LIN {X 0,Y 418.639,Z 217.334,A -85,B 0,C 180,E1 -10080,E2 -10080} C_VEL
LIN {X 0,Y 418.468,Z 217.355,A -85,B 0,C 180,E1 -10082.888,E2 -10082.888} C_VEL
LIN {X 0,Y 418.469,Z 217.355,A -85,B 0,C 180,E1 -10085.783,E2 -10085.783} C_VEL
LIN {X 0,Y 418.35,Z 217.368,A -85,B 0,C 180,E1 -10088.696,E2 -10088.696} C_VEL
LIN {X 0,Y 418.299,Z 217.373,A -85,B 0,C 180,E1 -10091.631,E2 -10091.631} C_VEL
LIN {X 0,Y 418.273,Z 217.382,A -85,B 0,C 180,E1 -10094.598,E2 -10094.598} C_VEL
LIN {X 0,Y 418.252,Z 217.38,A -85,B 0,C 180,E1 -10097.605,E2 -10097.605} C_VEL
LIN {X 0,Y 418.223,Z 217.388,A -85,B 0,C 180,E1 -10100.664,E2 -10100.664} C_VEL
LIN {X 0,Y 418.248,Z 217.383,A -85,B 0,C 180,E1 -10103.784,E2 -10103.784} C_VEL
LIN {X 0,Y 418.203,Z 217.392,A -85,B 0,C 180,E1 -10107.049,E2 -10107.049} C_VEL
LIN {X 0,Y 418.219,Z 217.385,A -85,B 0,C 180,E1 -10110.274,E2 -10110.274} C_VEL
LIN {X 0,Y 418.213,Z 217.383,A -85,B 0,C 180,E1 -10113.68,E2 -10113.68} C_VEL
LIN {X 0,Y 418.221,Z 217.379,A -85,B 0,C 180,E1 -10117.226,E2 -10117.226} C_VEL
LIN {X 0,Y 418.219,Z 217.379,A -85,B 0,C 180,E1 -10119.686,E2 -10119.686} C_VEL
LIN {X 0,Y 418.214,Z 217.391,A -85,B 0,C 180,E1 -10122.322,E2 -10122.322} C_VEL
LIN {X 0,Y 418.223,Z 217.385,A -85,B 0,C 180,E1 -10125.11,E2 -10125.11} C_VEL
LIN {X 0,Y 418.221,Z 217.386,A -85,B 0,C 180,E1 -10127.767,E2 -10127.767} C_VEL
LIN {X 0,Y 418.23,Z 217.385,A -85,B 0,C 180,E1 -10131.558,E2 -10131.558} C_VEL
LIN {X 0,Y 418.254,Z 217.383,A -85,B 0,C 180,E1 -10135.16,E2 -10135.16} C_VEL
LIN {X 0,Y 418.241,Z 217.384,A -85,B 0,C 180,E1 -10137.473,E2 -10137.473} C_VEL
LIN {X 0,Y 418.292,Z 217.381,A -85,B 0,C 180,E1 -10141.146,E2 -10141.146} C_VEL
LIN {X 0,Y 418.302,Z 217.657,A -85,B 0,C 180,E1 -10141.33,E2 -10141.33} C_VEL
LIN {X 0,Y 421.008,Z 229.949,A -85,B 0,C 180,E1 -10144.012,E2 -10144.012} C_VEL
LIN {X 0,Y 421.849,Z 235.282,A -85,B 0,C 180,E1 -10145.124,E2 -10145.124} C_VEL
LIN {X 0,Y 420.782,Z 249.932,A -85,B 0,C 180,E1 -10147.927,E2 -10147.927} C_VEL
LIN {X 0,Y 419.911,Z 263.738,A -85,B 0,C 180,E1 -10150.533,E2 -10150.533} C_VEL
LIN {X 0,Y 423.774,Z 286.188,A -85,B 0,C 180,E1 -10151.146,E2 -10151.146} C_VEL
LIN {X 0,Y 424.458,Z 292.992,A -85,B 0,C 180,E1 -10151.303,E2 -10151.303} C_VEL
LIN {X 0,Y 423.498,Z 373.222,A -85,B 0,C 180,E1 -10152.713,E2 -10152.713} C_VEL
LIN {X 0,Y 422.871,Z 386.948,A -85,B 0,C 180,E1 -10153.153,E2 -10153.153} C_VEL
LIN {X 0,Y 422.143,Z 399.294,A -85,B 0,C 180,E1 -10153.745,E2 -10153.745} C_VEL
LIN {X 0,Y 421.315,Z 411.136,A -85,B 0,C 180,E1 -10154.52,E2 -10154.52} C_VEL
LIN {X 0,Y 420.483,Z 422.531,A -85,B 0,C 180,E1 -10155.48,E2 -10155.48} C_VEL
LIN {X 0,Y 419.616,Z 432.832,A -85,B 0,C 180,E1 -10156.562,E2 -10156.562} C_VEL
LIN {X 0,Y 419.038,Z 441.272,A -85,B 0,C 180,E1 -10157.652,E2 -10157.652} C_VEL
LIN {X 0,Y 418.232,Z 450.447,A -85,B 0,C 180,E1 -10159.102,E2 -10159.102} C_VEL
LIN {X 0,Y 417.726,Z 457.856,A -85,B 0,C 180,E1 -10160.558,E2 -10160.558} C_VEL
LIN {X 0,Y 417.325,Z 464.7,A -85,B 0,C 180,E1 -10162.256,E2 -10162.256} C_VEL
LIN {X 0,Y 417.123,Z 469.362,A -85,B 0,C 180,E1 -10163.762,E2 -10163.762} C_VEL
LIN {X 0,Y 417.104,Z 472.691,A -85,B 0,C 180,E1 -10165.166,E2 -10165.166} C_VEL
LIN {X 0,Y 417.069,Z 475.74,A -85,B 0,C 180,E1 -10167.101,E2 -10167.101} C_VEL
LIN {X 0,Y 417.091,Z 476.67,A -85,B 0,C 180,E1 -10168.067,E2 -10168.067} C_VEL
LIN {X 0,Y 417.058,Z 477.19,A -85,B 0,C 180,E1 -10169.033,E2 -10169.033} C_VEL
LIN {X 0,Y 417.056,Z 477.282,A -85,B 0,C 180,E1 -10169.998,E2 -10169.998} C_VEL
LIN {X 0,Y 417.092,Z 476.305,A -85,B 0,C 180,E1 -10171.929,E2 -10171.929} C_VEL
LIN {X 0,Y 417.102,Z 475.215,A -85,B 0,C 180,E1 -10172.895,E2 -10172.895} C_VEL
LIN {X 0,Y 417.023,Z 473.664,A -85,B 0,C 180,E1 -10173.863,E2 -10173.863} C_VEL
LIN {X 0,Y 417.13,Z 470.551,A -85,B 0,C 180,E1 -10175.315,E2 -10175.315} C_VEL
LIN {X 0,Y 417.229,Z 466.36,A -85,B 0,C 180,E1 -10176.769,E2 -10176.769} C_VEL
LIN {X 0,Y 417.45,Z 459.955,A -85,B 0,C 180,E1 -10178.468,E2 -10178.468} C_VEL
LIN {X 0,Y 417.798,Z 452.974,A -85,B 0,C 180,E1 -10179.926,E2 -10179.926} C_VEL
LIN {X 0,Y 418.226,Z 445.837,A -85,B 0,C 180,E1 -10181.14,E2 -10181.14} C_VEL
LIN {X 0,Y 418.747,Z 437.203,A -85,B 0,C 180,E1 -10182.353,E2 -10182.353} C_VEL
LIN {X 0,Y 419.452,Z 426.544,A -85,B 0,C 180,E1 -10183.563,E2 -10183.563} C_VEL
LIN {X 0,Y 420.103,Z 415.971,A -85,B 0,C 180,E1 -10184.53,E2 -10184.53} C_VEL
LIN {X 0,Y 420.782,Z 404.288,A -85,B 0,C 180,E1 -10185.372,E2 -10185.372} C_VEL
LIN {X 0,Y 421.426,Z 392.137,A -85,B 0,C 180,E1 -10186.031,E2 -10186.031} C_VEL
LIN {X 0,Y 421.967,Z 379.849,A -85,B 0,C 180,E1 -10186.506,E2 -10186.506} C_VEL
LIN {X 0,Y 422.292,Z 366.152,A -85,B 0,C 180,E1 -10186.835,E2 -10186.835} C_VEL
LIN {X 0,Y 422.863,Z 289.846,A -85,B 0,C 180,E1 -10188.135,E2 -10188.135} C_VEL
LIN {X 0,Y 419.286,Z 264.116,A -85,B 0,C 180,E1 -10188.725,E2 -10188.725} C_VEL
LIN {X 0,Y 420.277,Z 245.887,A -85,B 0,C 180,E1 -10192.097,E2 -10192.097} C_VEL
LIN {X 0,Y 421.029,Z 232.178,A -85,B 0,C 180,E1 -10194.66,E2 -10194.66} C_VEL
LIN {X 0,Y 419.604,Z 223.737,A -85,B 0,C 180,E1 -10196.345,E2 -10196.345} C_VEL
LIN {X 0,Y 418.339,Z 217.378,A -85,B 0,C 180,E1 -10197.69,E2 -10197.69} C_VEL
LIN {X 0,Y 418.195,Z 217.393,A -85,B 0,C 180,E1 -10201.392,E2 -10201.392} C_VEL
LIN {X 0,Y 418.246,Z 217.384,A -85,B 0,C 180,E1 -10204.576,E2 -10204.576} C_VEL
LIN {X 0,Y 418.205,Z 217.393,A -85,B 0,C 180,E1 -10207.829,E2 -10207.829} C_VEL
LIN {X 0,Y 418.196,Z 217.389,A -85,B 0,C 180,E1 -10210.944,E2 -10210.944} C_VEL
LIN {X 0,Y 418.182,Z 217.396,A -85,B 0,C 180,E1 -10213.725,E2 -10213.725} C_VEL
LIN {X 0,Y 418.231,Z 217.385,A -85,B 0,C 180,E1 -10216.451,E2 -10216.451} C_VEL
LIN {X 0,Y 418.234,Z 217.385,A -85,B 0,C 180,E1 -10219.119,E2 -10219.119} C_VEL
LIN {X 0,Y 418.202,Z 217.39,A -85,B 0,C 180,E1 -10222.161,E2 -10222.161} C_VEL
LIN {X 0,Y 418.226,Z 217.389,A -85,B 0,C 180,E1 -10225.416,E2 -10225.416} C_VEL
LIN {X 0,Y 418.173,Z 217.391,A -85,B 0,C 180,E1 -10228.601,E2 -10228.601} C_VEL
LIN {X 0,Y 418.251,Z 217.385,A -85,B 0,C 180,E1 -10231.934,E2 -10231.934} C_VEL
LIN {X 0,Y 418.245,Z 217.386,A -85,B 0,C 180,E1 -10235.16,E2 -10235.16} C_VEL
LIN {X 0,Y 418.225,Z 217.385,A -85,B 0,C 180,E1 -10238.303,E2 -10238.303} C_VEL
LIN {X 0,Y 418.239,Z 217.391,A -85,B 0,C 180,E1 -10241.381,E2 -10241.381} C_VEL
LIN {X 0,Y 418.259,Z 217.381,A -85,B 0,C 180,E1 -10244.404,E2 -10244.404} C_VEL
LIN {X 0,Y 418.319,Z 217.379,A -85,B 0,C 180,E1 -10247.385,E2 -10247.385} C_VEL
LIN {X 0,Y 418.364,Z 217.374,A -85,B 0,C 180,E1 -10251.304,E2 -10251.304} C_VEL
LIN {X 0,Y 418.486,Z 217.352,A -85,B 0,C 180,E1 -10254.217,E2 -10254.217} C_VEL
LIN {X 0,Y 418.489,Z 217.352,A -85,B 0,C 180,E1 -10258.075,E2 -10258.075} C_VEL
LIN {X 0,Y 418.616,Z 217.336,A -85,B 0,C 180,E1 -10260,E2 -10260} C_VEL
LIN {X 0,Y 418.446,Z 217.364,A -85,B 0,C 180,E1 -10262.888,E2 -10262.888} C_VEL
LIN {X 0,Y 418.435,Z 217.364,A -85,B 0,C 180,E1 -10266.752,E2 -10266.752} C_VEL
LIN {X 0,Y 418.292,Z 217.377,A -85,B 0,C 180,E1 -10269.673,E2 -10269.673} C_VEL
LIN {X 0,Y 418.304,Z 217.38,A -85,B 0,C 180,E1 -10273.007,E2 -10273.007} C_VEL
LIN {X 0,Y 418.269,Z 217.387,A -85,B 0,C 180,E1 -10276.74,E2 -10276.74} C_VEL
LIN {X 0,Y 418.221,Z 217.386,A -85,B 0,C 180,E1 -10279.792,E2 -10279.792} C_VEL
LIN {X 0,Y 418.185,Z 217.396,A -85,B 0,C 180,E1 -10282.739,E2 -10282.739} C_VEL
LIN {X 0,Y 418.225,Z 217.386,A -85,B 0,C 180,E1 -10285.907,E2 -10285.907} C_VEL
LIN {X 0,Y 418.231,Z 217.385,A -85,B 0,C 180,E1 -10289.165,E2 -10289.165} C_VEL
LIN {X 0,Y 418.217,Z 217.389,A -85,B 0,C 180,E1 -10292.847,E2 -10292.847} C_VEL
LIN {X 0,Y 418.208,Z 217.392,A -85,B 0,C 180,E1 -10296.242,E2 -10296.242} C_VEL
LIN {X 0,Y 418.228,Z 217.385,A -85,B 0,C 180,E1 -10299.685,E2 -10299.685} C_VEL
LIN {X 0,Y 418.252,Z 217.389,A -85,B 0,C 180,E1 -10302.333,E2 -10302.333} C_VEL
LIN {X 0,Y 418.217,Z 217.386,A -85,B 0,C 180,E1 -10305.114,E2 -10305.114} C_VEL
LIN {X 0,Y 418.214,Z 217.389,A -85,B 0,C 180,E1 -10307.771,E2 -10307.771} C_VEL
LIN {X 0,Y 418.234,Z 217.386,A -85,B 0,C 180,E1 -10310.623,E2 -10310.623} C_VEL
LIN {X 0,Y 418.223,Z 217.391,A -85,B 0,C 180,E1 -10313.98,E2 -10313.98} C_VEL
LIN {X 0,Y 418.24,Z 217.383,A -85,B 0,C 180,E1 -10317.16,E2 -10317.16} C_VEL
LIN {X 0,Y 418.255,Z 217.381,A -85,B 0,C 180,E1 -10320.9,E2 -10320.9} C_VEL
LIN {X 0,Y 418.257,Z 217.386,A -85,B 0,C 180,E1 -10324.1,E2 -10324.1} C_VEL
LIN {X 0,Y 418.223,Z 217.386,A -85,B 0,C 180,E1 -10327.267,E2 -10327.267} C_VEL
LIN {X 0,Y 418.277,Z 217.38,A -85,B 0,C 180,E1 -10330.368,E2 -10330.368} C_VEL
LIN {X 0,Y 418.312,Z 217.377,A -85,B 0,C 180,E1 -10333.408,E2 -10333.408} C_VEL
LIN {X 0,Y 418.345,Z 217.371,A -85,B 0,C 180,E1 -10337.002,E2 -10337.002} C_VEL
LIN {X 0,Y 418.362,Z 217.476,A -85,B 0,C 180,E1 -10339.996,E2 -10339.996} C_VEL
LIN {X 0,Y 419.753,Z 225.468,A -85,B 0,C 180,E1 -10341.821,E2 -10341.821} C_VEL
LIN {X 0,Y 419.713,Z 228.011,A -85,B 0,C 180,E1 -10342.371,E2 -10342.371} C_VEL
LIN {X 0,Y 423.404,Z 248.524,A -85,B 0,C 180,E1 -10342.881,E2 -10342.881} C_VEL
LIN {X 0,Y 422.273,Z 335.092,A -85,B 0,C 180,E1 -10344.361,E2 -10344.361} C_VEL
LIN {X 0,Y 421.932,Z 348.28,A -85,B 0,C 180,E1 -10344.776,E2 -10344.776} C_VEL
LIN {X 0,Y 421.84,Z 354.693,A -85,B 0,C 180,E1 -10345.056,E2 -10345.056} C_VEL
LIN {X 0,Y 420.996,Z 360.232,A -85,B 0,C 180,E1 -10345.312,E2 -10345.312} C_VEL
LIN {X 0,Y 417.843,Z 369.054,A -85,B 0,C 180,E1 -10345.756,E2 -10345.756} C_VEL
LIN {X 0,Y 414.563,Z 377.579,A -85,B 0,C 180,E1 -10346.292,E2 -10346.292} C_VEL
LIN {X 0,Y 413.511,Z 382.59,A -85,B 0,C 180,E1 -10346.701,E2 -10346.701} C_VEL
LIN {X 0,Y 412.792,Z 393.404,A -85,B 0,C 180,E1 -10347.807,E2 -10347.807} C_VEL
LIN {X 0,Y 412.144,Z 403.005,A -85,B 0,C 180,E1 -10349.025,E2 -10349.025} C_VEL
LIN {X 0,Y 411.629,Z 410.879,A -85,B 0,C 180,E1 -10350.246,E2 -10350.246} C_VEL
LIN {X 0,Y 411.019,Z 418.618,A -85,B 0,C 180,E1 -10351.716,E2 -10351.716} C_VEL
LIN {X 0,Y 410.69,Z 425.692,A -85,B 0,C 180,E1 -10353.435,E2 -10353.435} C_VEL
LIN {X 0,Y 410.351,Z 430.439,A -85,B 0,C 180,E1 -10354.914,E2 -10354.914} C_VEL
LIN {X 0,Y 410.226,Z 434.196,A -85,B 0,C 180,E1 -10356.453,E2 -10356.453} C_VEL
LIN {X 0,Y 410.057,Z 436.704,A -85,B 0,C 180,E1 -10357.882,E2 -10357.882} C_VEL
LIN {X 0,Y 409.974,Z 437.947,A -85,B 0,C 180,E1 -10358.876,E2 -10358.876} C_VEL
LIN {X 0,Y 409.907,Z 438.765,A -85,B 0,C 180,E1 -10359.873,E2 -10359.873} C_VEL
LIN {X 0,Y 409.966,Z 439.155,A -85,B 0,C 180,E1 -10360.87,E2 -10360.87} C_VEL
LIN {X 0,Y 410,Z 439.052,A -85,B 0,C 180,E1 -10362.294,E2 -10362.294} C_VEL
LIN {X 0,Y 410.021,Z 437.952,A -85,B 0,C 180,E1 -10363.885,E2 -10363.885} C_VEL
LIN {X 0,Y 410.108,Z 436.698,A -85,B 0,C 180,E1 -10364.896,E2 -10364.896} C_VEL
LIN {X 0,Y 410.413,Z 433.881,A -85,B 0,C 180,E1 -10366.471,E2 -10366.471} C_VEL
LIN {X 0,Y 410.681,Z 430.238,A -85,B 0,C 180,E1 -10367.941,E2 -10367.941} C_VEL
LIN {X 0,Y 411.096,Z 425.31,A -85,B 0,C 180,E1 -10369.464,E2 -10369.464} C_VEL
LIN {X 0,Y 411.684,Z 418.963,A -85,B 0,C 180,E1 -10371.008,E2 -10371.008} C_VEL
LIN {X 0,Y 412.304,Z 412.445,A -85,B 0,C 180,E1 -10372.288,E2 -10372.288} C_VEL
LIN {X 0,Y 413.037,Z 404.552,A -85,B 0,C 180,E1 -10373.569,E2 -10373.569} C_VEL
LIN {X 0,Y 413.863,Z 394.792,A -85,B 0,C 180,E1 -10374.852,E2 -10374.852} C_VEL
LIN {X 0,Y 414.764,Z 384.155,A -85,B 0,C 180,E1 -10375.974,E2 -10375.974} C_VEL
LIN {X 0,Y 415.548,Z 373.203,A -85,B 0,C 180,E1 -10376.898,E2 -10376.898} C_VEL
LIN {X 0,Y 416.144,Z 361.394,A -85,B 0,C 180,E1 -10377.672,E2 -10377.672} C_VEL
LIN {X 0,Y 416.778,Z 348.137,A -85,B 0,C 180,E1 -10378.301,E2 -10378.301} C_VEL
LIN {X 0,Y 417.168,Z 334.958,A -85,B 0,C 180,E1 -10378.713,E2 -10378.713} C_VEL
LIN {X 0,Y 418.332,Z 247.723,A -85,B 0,C 180,E1 -10380.255,E2 -10380.255} C_VEL
LIN {X 0,Y 414.124,Z 230.945,A -85,B 0,C 180,E1 -10380.806,E2 -10380.806} C_VEL
LIN {X 0,Y 413.352,Z 228.534,A -85,B 0,C 180,E1 -10380.923,E2 -10380.923} C_VEL
LIN {X 0,Y 411.227,Z 218.261,A -85,B 0,C 180,E1 -10383.445,E2 -10383.445} C_VEL
LIN {X 0,Y 411.188,Z 218.268,A -85,B 0,C 180,E1 -10386.74,E2 -10386.74} C_VEL
LIN {X 0,Y 411.219,Z 218.263,A -85,B 0,C 180,E1 -10389.728,E2 -10389.728} C_VEL
LIN {X 0,Y 411.168,Z 218.268,A -85,B 0,C 180,E1 -10393.131,E2 -10393.131} C_VEL
LIN {X 0,Y 411.21,Z 218.265,A -85,B 0,C 180,E1 -10395.872,E2 -10395.872} C_VEL
LIN {X 0,Y 411.197,Z 218.264,A -85,B 0,C 180,E1 -10398.763,E2 -10398.763} C_VEL
LIN {X 0,Y 411.188,Z 218.265,A -85,B 0,C 180,E1 -10402.025,E2 -10402.025} C_VEL
LIN {X 0,Y 411.189,Z 218.264,A -85,B 0,C 180,E1 -10405.665,E2 -10405.665} C_VEL
LIN {X 0,Y 411.178,Z 218.261,A -85,B 0,C 180,E1 -10409.151,E2 -10409.151} C_VEL
LIN {X 0,Y 411.24,Z 218.252,A -85,B 0,C 180,E1 -10412.521,E2 -10412.521} C_VEL
LIN {X 0,Y 411.199,Z 218.261,A -85,B 0,C 180,E1 -10415.783,E2 -10415.783} C_VEL
LIN {X 0,Y 411.172,Z 218.265,A -85,B 0,C 180,E1 -10418.964,E2 -10418.964} C_VEL
LIN {X 0,Y 411.228,Z 218.259,A -85,B 0,C 180,E1 -10422.084,E2 -10422.084} C_VEL
LIN {X 0,Y 411.236,Z 218.253,A -85,B 0,C 180,E1 -10425.146,E2 -10425.146} C_VEL
LIN {X 0,Y 411.256,Z 218.252,A -85,B 0,C 180,E1 -10428.166,E2 -10428.166} C_VEL
LIN {X 0,Y 411.418,Z 218.233,A -85,B 0,C 180,E1 -10432.185,E2 -10432.185} C_VEL
LIN {X 0,Y 411.451,Z 218.227,A -85,B 0,C 180,E1 -10434.118,E2 -10434.118} C_VEL
LIN {X 0,Y 411.48,Z 218.22,A -85,B 0,C 180,E1 -10438.042,E2 -10438.042} C_VEL
LIN {X 0,Y 411.61,Z 218.21,A -85,B 0,C 180,E1 -10440,E2 -10440} C_VEL
LIN {X 0,Y 411.425,Z 218.232,A -85,B 0,C 180,E1 -10442.937,E2 -10442.937} C_VEL
LIN {X 0,Y 411.402,Z 218.237,A -85,B 0,C 180,E1 -10446.868,E2 -10446.868} C_VEL
LIN {X 0,Y 411.267,Z 218.252,A -85,B 0,C 180,E1 -10449.839,E2 -10449.839} C_VEL
LIN {X 0,Y 411.283,Z 218.251,A -85,B 0,C 180,E1 -10453.106,E2 -10453.106} C_VEL
LIN {X 0,Y 411.243,Z 218.254,A -85,B 0,C 180,E1 -10456.889,E2 -10456.889} C_VEL
LIN {X 0,Y 411.186,Z 218.263,A -85,B 0,C 180,E1 -10459.989,E2 -10459.989} C_VEL
LIN {X 0,Y 411.171,Z 218.267,A -85,B 0,C 180,E1 -10463.149,E2 -10463.149} C_VEL
LIN {X 0,Y 411.165,Z 218.263,A -85,B 0,C 180,E1 -10466.386,E2 -10466.386} C_VEL
LIN {X 0,Y 411.176,Z 218.26,A -85,B 0,C 180,E1 -10469.715,E2 -10469.715} C_VEL
LIN {X 0,Y 411.186,Z 218.259,A -85,B 0,C 180,E1 -10473.158,E2 -10473.158} C_VEL
LIN {X 0,Y 411.175,Z 218.262,A -85,B 0,C 180,E1 -10476.554,E2 -10476.554} C_VEL
LIN {X 0,Y 411.185,Z 218.255,A -85,B 0,C 180,E1 -10479.727,E2 -10479.727} C_VEL
LIN {X 0,Y 411.159,Z 218.266,A -85,B 0,C 180,E1 -10483.136,E2 -10483.136} C_VEL
LIN {X 0,Y 411.156,Z 218.268,A -85,B 0,C 180,E1 -10485.883,E2 -10485.883} C_VEL
LIN {X 0,Y 411.143,Z 218.267,A -85,B 0,C 180,E1 -10488.775,E2 -10488.775} C_VEL
LIN {X 0,Y 411.179,Z 218.263,A -85,B 0,C 180,E1 -10492.027,E2 -10492.027} C_VEL
LIN {X 0,Y 411.201,Z 218.265,A -85,B 0,C 180,E1 -10495.668,E2 -10495.668} C_VEL
LIN {X 0,Y 411.186,Z 218.267,A -85,B 0,C 180,E1 -10499.153,E2 -10499.153} C_VEL
LIN {X 0,Y 411.247,Z 218.297,A -85,B 0,C 180,E1 -10500.932,E2 -10500.932} C_VEL
LIN {X 0,Y 414.089,Z 231.233,A -85,B 0,C 180,E1 -10503.815,E2 -10503.815} C_VEL
LIN {X 0,Y 414.974,Z 236.561,A -85,B 0,C 180,E1 -10504.951,E2 -10504.951} C_VEL
LIN {X 0,Y 413.866,Z 251.201,A -85,B 0,C 180,E1 -10507.801,E2 -10507.801} C_VEL
LIN {X 0,Y 413.06,Z 263.345,A -85,B 0,C 180,E1 -10510.138,E2 -10510.138} C_VEL
LIN {X 0,Y 417.187,Z 287.154,A -85,B 0,C 180,E1 -10510.811,E2 -10510.811} C_VEL
LIN {X 0,Y 417.832,Z 294.371,A -85,B 0,C 180,E1 -10510.977,E2 -10510.977} C_VEL
LIN {X 0,Y 416.85,Z 372.337,A -85,B 0,C 180,E1 -10512.365,E2 -10512.365} C_VEL
LIN {X 0,Y 416.249,Z 385.481,A -85,B 0,C 180,E1 -10512.782,E2 -10512.782} C_VEL
LIN {X 0,Y 415.49,Z 397.575,A -85,B 0,C 180,E1 -10513.351,E2 -10513.351} C_VEL
LIN {X 0,Y 414.587,Z 409.813,A -85,B 0,C 180,E1 -10514.136,E2 -10514.136} C_VEL
LIN {X 0,Y 413.709,Z 421.384,A -85,B 0,C 180,E1 -10515.111,E2 -10515.111} C_VEL
LIN {X 0,Y 412.805,Z 431.82,A -85,B 0,C 180,E1 -10516.21,E2 -10516.21} C_VEL
LIN {X 0,Y 412.085,Z 441.247,A -85,B 0,C 180,E1 -10517.44,E2 -10517.44} C_VEL
LIN {X 0,Y 411.249,Z 450.358,A -85,B 0,C 180,E1 -10518.915,E2 -10518.915} C_VEL
LIN {X 0,Y 410.701,Z 457.722,A -85,B 0,C 180,E1 -10520.395,E2 -10520.395} C_VEL
LIN {X 0,Y 410.267,Z 464.51,A -85,B 0,C 180,E1 -10522.122,E2 -10522.122} C_VEL
LIN {X 0,Y 410.043,Z 469.447,A -85,B 0,C 180,E1 -10523.775,E2 -10523.775} C_VEL
LIN {X 0,Y 410.012,Z 472.437,A -85,B 0,C 180,E1 -10525.082,E2 -10525.082} C_VEL
LIN {X 0,Y 409.966,Z 475.458,A -85,B 0,C 180,E1 -10527.05,E2 -10527.05} C_VEL
LIN {X 0,Y 410.018,Z 476.376,A -85,B 0,C 180,E1 -10528.034,E2 -10528.034} C_VEL
LIN {X 0,Y 409.98,Z 476.869,A -85,B 0,C 180,E1 -10529.016,E2 -10529.016} C_VEL
LIN {X 0,Y 409.976,Z 476.948,A -85,B 0,C 180,E1 -10529.998,E2 -10529.998} C_VEL
LIN {X 0,Y 410.02,Z 475.945,A -85,B 0,C 180,E1 -10531.963,E2 -10531.963} C_VEL
LIN {X 0,Y 410,Z 474.828,A -85,B 0,C 180,E1 -10532.946,E2 -10532.946} C_VEL
LIN {X 0,Y 409.942,Z 473.261,A -85,B 0,C 180,E1 -10533.93,E2 -10533.93} C_VEL
LIN {X 0,Y 410.025,Z 470.116,A -85,B 0,C 180,E1 -10535.407,E2 -10535.407} C_VEL
LIN {X 0,Y 410.16,Z 465.895,A -85,B 0,C 180,E1 -10536.886,E2 -10536.886} C_VEL
LIN {X 0,Y 410.377,Z 459.453,A -85,B 0,C 180,E1 -10538.616,E2 -10538.616} C_VEL
LIN {X 0,Y 410.736,Z 452.422,A -85,B 0,C 180,E1 -10540.098,E2 -10540.098} C_VEL
LIN {X 0,Y 411.326,Z 443.601,A -85,B 0,C 180,E1 -10541.579,E2 -10541.579} C_VEL
LIN {X 0,Y 411.917,Z 434.557,A -85,B 0,C 180,E1 -10542.812,E2 -10542.812} C_VEL
LIN {X 0,Y 412.601,Z 424.611,A -85,B 0,C 180,E1 -10543.918,E2 -10543.918} C_VEL
LIN {X 0,Y 413.285,Z 413.595,A -85,B 0,C 180,E1 -10544.901,E2 -10544.901} C_VEL
LIN {X 0,Y 414.057,Z 401.237,A -85,B 0,C 180,E1 -10545.755,E2 -10545.755} C_VEL
LIN {X 0,Y 414.688,Z 388.182,A -85,B 0,C 180,E1 -10546.425,E2 -10546.425} C_VEL
LIN {X 0,Y 415.212,Z 374.897,A -85,B 0,C 180,E1 -10546.878,E2 -10546.878} C_VEL
LIN {X 0,Y 415.54,Z 354.224,A -85,B 0,C 180,E1 -10547.276,E2 -10547.276} C_VEL
LIN {X 0,Y 416.04,Z 290.792,A -85,B 0,C 180,E1 -10548.374,E2 -10548.374} C_VEL
LIN {X 0,Y 412.325,Z 263.698,A -85,B 0,C 180,E1 -10549.021,E2 -10549.021} C_VEL
LIN {X 0,Y 413.471,Z 243.924,A -85,B 0,C 180,E1 -10552.745,E2 -10552.745} C_VEL
LIN {X 0,Y 414.039,Z 232.94,A -85,B 0,C 180,E1 -10554.837,E2 -10554.837} C_VEL
LIN {X 0,Y 411.874,Z 221.104,A -85,B 0,C 180,E1 -10557.261,E2 -10557.261} C_VEL
LIN {X 0,Y 411.296,Z 218.255,A -85,B 0,C 180,E1 -10557.884,E2 -10557.884} C_VEL
LIN {X 0,Y 411.165,Z 218.268,A -85,B 0,C 180,E1 -10561.279,E2 -10561.279} C_VEL
LIN {X 0,Y 411.187,Z 218.265,A -85,B 0,C 180,E1 -10564.329,E2 -10564.329} C_VEL
LIN {X 0,Y 411.171,Z 218.271,A -85,B 0,C 180,E1 -10567.97,E2 -10567.97} C_VEL
LIN {X 0,Y 411.137,Z 218.269,A -85,B 0,C 180,E1 -10571.224,E2 -10571.224} C_VEL
LIN {X 0,Y 411.152,Z 218.267,A -85,B 0,C 180,E1 -10574.486,E2 -10574.486} C_VEL
LIN {X 0,Y 411.196,Z 218.262,A -85,B 0,C 180,E1 -10577.293,E2 -10577.293} C_VEL
LIN {X 0,Y 411.197,Z 218.26,A -85,B 0,C 180,E1 -10580.773,E2 -10580.773} C_VEL
LIN {X 0,Y 411.161,Z 218.265,A -85,B 0,C 180,E1 -10584.467,E2 -10584.467} C_VEL
LIN {X 0,Y 411.168,Z 218.264,A -85,B 0,C 180,E1 -10586.87,E2 -10586.87} C_VEL
LIN {X 0,Y 411.198,Z 218.26,A -85,B 0,C 180,E1 -10590.639,E2 -10590.639} C_VEL
LIN {X 0,Y 411.195,Z 218.267,A -85,B 0,C 180,E1 -10593.616,E2 -10593.616} C_VEL
LIN {X 0,Y 411.225,Z 218.263,A -85,B 0,C 180,E1 -10597.333,E2 -10597.333} C_VEL
LIN {X 0,Y 411.219,Z 218.259,A -85,B 0,C 180,E1 -10600.028,E2 -10600.028} C_VEL
LIN {X 0,Y 411.215,Z 218.263,A -85,B 0,C 180,E1 -10603.129,E2 -10603.129} C_VEL
LIN {X 0,Y 411.262,Z 218.255,A -85,B 0,C 180,E1 -10606.89,E2 -10606.89} C_VEL
LIN {X 0,Y 411.261,Z 218.253,A -85,B 0,C 180,E1 -10610.161,E2 -10610.161} C_VEL
LIN {X 0,Y 411.425,Z 218.239,A -85,B 0,C 180,E1 -10613.133,E2 -10613.133} C_VEL
LIN {X 0,Y 411.264,Z 218.259,A -85,B 0,C 180,E1 -10615.099,E2 -10615.099} C_VEL
LIN {X 0,Y 411.459,Z 218.228,A -85,B 0,C 180,E1 -10618.042,E2 -10618.042} C_VEL
LIN {X 0,Y 411.586,Z 218.212,A -85,B 0,C 180,E1 -10620,E2 -10620} C_VEL
LIN {X 0,Y 411.403,Z 218.241,A -85,B 0,C 180,E1 -10622.938,E2 -10622.938} C_VEL
LIN {X 0,Y 411.403,Z 218.242,A -85,B 0,C 180,E1 -10626.868,E2 -10626.868} C_VEL
LIN {X 0,Y 411.245,Z 218.255,A -85,B 0,C 180,E1 -10629.84,E2 -10629.84} C_VEL
LIN {X 0,Y 411.263,Z 218.256,A -85,B 0,C 180,E1 -10633.11,E2 -10633.11} C_VEL
LIN {X 0,Y 411.212,Z 218.264,A -85,B 0,C 180,E1 -10636.891,E2 -10636.891} C_VEL
LIN {X 0,Y 411.162,Z 218.265,A -85,B 0,C 180,E1 -10639.99,E2 -10639.99} C_VEL
LIN {X 0,Y 411.15,Z 218.268,A -85,B 0,C 180,E1 -10643.151,E2 -10643.151} C_VEL
LIN {X 0,Y 411.194,Z 218.266,A -85,B 0,C 180,E1 -10646.384,E2 -10646.384} C_VEL
LIN {X 0,Y 411.168,Z 218.264,A -85,B 0,C 180,E1 -10649.716,E2 -10649.716} C_VEL
LIN {X 0,Y 411.168,Z 218.265,A -85,B 0,C 180,E1 -10653.16,E2 -10653.16} C_VEL
LIN {X 0,Y 411.156,Z 218.271,A -85,B 0,C 180,E1 -10656.556,E2 -10656.556} C_VEL
LIN {X 0,Y 411.191,Z 218.262,A -85,B 0,C 180,E1 -10659.734,E2 -10659.734} C_VEL
LIN {X 0,Y 411.187,Z 218.262,A -85,B 0,C 180,E1 -10663.132,E2 -10663.132} C_VEL
LIN {X 0,Y 411.143,Z 218.27,A -85,B 0,C 180,E1 -10665.885,E2 -10665.885} C_VEL
LIN {X 0,Y 411.139,Z 218.269,A -85,B 0,C 180,E1 -10668.776,E2 -10668.776} C_VEL
LIN {X 0,Y 411.184,Z 218.266,A -85,B 0,C 180,E1 -10671.836,E2 -10671.836} C_VEL
LIN {X 0,Y 411.192,Z 218.261,A -85,B 0,C 180,E1 -10675.126,E2 -10675.126} C_VEL
LIN {X 0,Y 411.149,Z 218.274,A -85,B 0,C 180,E1 -10678.007,E2 -10678.007} C_VEL
LIN {X 0,Y 411.204,Z 218.261,A -85,B 0,C 180,E1 -10681.414,E2 -10681.414} C_VEL
LIN {X 0,Y 411.225,Z 218.261,A -85,B 0,C 180,E1 -10683.623,E2 -10683.623} C_VEL
LIN {X 0,Y 411.187,Z 218.262,A -85,B 0,C 180,E1 -10686.856,E2 -10686.856} C_VEL
LIN {X 0,Y 411.208,Z 218.263,A -85,B 0,C 180,E1 -10690.054,E2 -10690.054} C_VEL
LIN {X 0,Y 411.259,Z 218.254,A -85,B 0,C 180,E1 -10693.135,E2 -10693.135} C_VEL
LIN {X 0,Y 411.304,Z 218.247,A -85,B 0,C 180,E1 -10696.899,E2 -10696.899} C_VEL
LIN {X 0,Y 411.289,Z 218.281,A -85,B 0,C 180,E1 -10699.791,E2 -10699.791} C_VEL
LIN {X 0,Y 412.79,Z 227.061,A -85,B 0,C 180,E1 -10701.822,E2 -10701.822} C_VEL
LIN {X 0,Y 412.784,Z 228.347,A -85,B 0,C 180,E1 -10702.103,E2 -10702.103} C_VEL
LIN {X 0,Y 416.563,Z 248.374,A -85,B 0,C 180,E1 -10702.611,E2 -10702.611} C_VEL
LIN {X 0,Y 415.433,Z 336.2,A -85,B 0,C 180,E1 -10704.146,E2 -10704.146} C_VEL
LIN {X 0,Y 415.025,Z 349.897,A -85,B 0,C 180,E1 -10704.597,E2 -10704.597} C_VEL
LIN {X 0,Y 414.582,Z 362.183,A -85,B 0,C 180,E1 -10705.201,E2 -10705.201} C_VEL
LIN {X 0,Y 414.109,Z 373.942,A -85,B 0,C 180,E1 -10705.988,E2 -10705.988} C_VEL
LIN {X 0,Y 413.511,Z 382.59,A -85,B 0,C 180,E1 -10706.701,E2 -10706.701} C_VEL
LIN {X 0,Y 412.449,Z 387.494,A -85,B 0,C 180,E1 -10707.139,E2 -10707.139} C_VEL
LIN {X 0,Y 409.071,Z 395.155,A -85,B 0,C 180,E1 -10707.887,E2 -10707.887} C_VEL
LIN {X 0,Y 405.808,Z 402.316,A -85,B 0,C 180,E1 -10708.735,E2 -10708.735} C_VEL
LIN {X 0,Y 404.931,Z 406.409,A -85,B 0,C 180,E1 -10709.322,E2 -10709.322} C_VEL
LIN {X 0,Y 404.355,Z 414.744,A -85,B 0,C 180,E1 -10710.749,E2 -10710.749} C_VEL
LIN {X 0,Y 403.843,Z 421.787,A -85,B 0,C 180,E1 -10712.246,E2 -10712.246} C_VEL
LIN {X 0,Y 403.506,Z 428.202,A -85,B 0,C 180,E1 -10713.996,E2 -10713.996} C_VEL
LIN {X 0,Y 403.26,Z 432.454,A -85,B 0,C 180,E1 -10715.502,E2 -10715.502} C_VEL
LIN {X 0,Y 403.056,Z 435.653,A -85,B 0,C 180,E1 -10717.012,E2 -10717.012} C_VEL
LIN {X 0,Y 402.96,Z 437.247,A -85,B 0,C 180,E1 -10718.022,E2 -10718.022} C_VEL
LIN {X 0,Y 402.867,Z 438.429,A -85,B 0,C 180,E1 -10719.034,E2 -10719.034} C_VEL
LIN {X 0,Y 402.883,Z 439.509,A -85,B 0,C 180,E1 -10721.064,E2 -10721.064} C_VEL
LIN {X 0,Y 402.932,Z 439.373,A -85,B 0,C 180,E1 -10722.375,E2 -10722.375} C_VEL
LIN {X 0,Y 402.947,Z 438.114,A -85,B 0,C 180,E1 -10724.134,E2 -10724.134} C_VEL
LIN {X 0,Y 403.076,Z 436.81,A -85,B 0,C 180,E1 -10725.162,E2 -10725.162} C_VEL
LIN {X 0,Y 403.378,Z 434.213,A -85,B 0,C 180,E1 -10726.612,E2 -10726.612} C_VEL
LIN {X 0,Y 403.696,Z 430.14,A -85,B 0,C 180,E1 -10728.262,E2 -10728.262} C_VEL
LIN {X 0,Y 404.145,Z 425.384,A -85,B 0,C 180,E1 -10729.73,E2 -10729.73} C_VEL
LIN {X 0,Y 404.795,Z 418.602,A -85,B 0,C 180,E1 -10731.383,E2 -10731.383} C_VEL
LIN {X 0,Y 405.633,Z 410.532,A -85,B 0,C 180,E1 -10732.924,E2 -10732.924} C_VEL
LIN {X 0,Y 406.421,Z 401.988,A -85,B 0,C 180,E1 -10734.248,E2 -10734.248} C_VEL
LIN {X 0,Y 407.341,Z 391.575,A -85,B 0,C 180,E1 -10735.552,E2 -10735.552} C_VEL
LIN {X 0,Y 408.278,Z 381.135,A -85,B 0,C 180,E1 -10736.586,E2 -10736.586} C_VEL
LIN {X 0,Y 409.074,Z 369.623,A -85,B 0,C 180,E1 -10737.497,E2 -10737.497} C_VEL
LIN {X 0,Y 409.697,Z 357.839,A -85,B 0,C 180,E1 -10738.216,E2 -10738.216} C_VEL
LIN {X 0,Y 410.242,Z 345.167,A -85,B 0,C 180,E1 -10738.765,E2 -10738.765} C_VEL
LIN {X 0,Y 410.609,Z 332.42,A -85,B 0,C 180,E1 -10739.118,E2 -10739.118} C_VEL
LIN {X 0,Y 411.785,Z 249.064,A -85,B 0,C 180,E1 -10740.606,E2 -10740.606} C_VEL
LIN {X 0,Y 407.9,Z 233.47,A -85,B 0,C 180,E1 -10741.13,E2 -10741.13} C_VEL
LIN {X 0,Y 406.258,Z 228.88,A -85,B 0,C 180,E1 -10741.343,E2 -10741.343} C_VEL
LIN {X 0,Y 404.197,Z 219.136,A -85,B 0,C 180,E1 -10743.806,E2 -10743.806} C_VEL
LIN {X 0,Y 404.143,Z 219.146,A -85,B 0,C 180,E1 -10747.49,E2 -10747.49} C_VEL
LIN {X 0,Y 404.158,Z 219.14,A -85,B 0,C 180,E1 -10750.081,E2 -10750.081} C_VEL
LIN {X 0,Y 404.149,Z 219.142,A -85,B 0,C 180,E1 -10753.083,E2 -10753.083} C_VEL
LIN {X 0,Y 404.185,Z 219.141,A -85,B 0,C 180,E1 -10755.931,E2 -10755.931} C_VEL
LIN {X 0,Y 404.151,Z 219.142,A -85,B 0,C 180,E1 -10758.639,E2 -10758.639} C_VEL
LIN {X 0,Y 404.147,Z 219.143,A -85,B 0,C 180,E1 -10761.489,E2 -10761.489} C_VEL
LIN {X 0,Y 404.169,Z 219.137,A -85,B 0,C 180,E1 -10764.982,E2 -10764.982} C_VEL
LIN {X 0,Y 404.126,Z 219.14,A -85,B 0,C 180,E1 -10768.552,E2 -10768.552} C_VEL
LIN {X 0,Y 404.178,Z 219.135,A -85,B 0,C 180,E1 -10771.999,E2 -10771.999} C_VEL
LIN {X 0,Y 404.154,Z 219.142,A -85,B 0,C 180,E1 -10775.333,E2 -10775.333} C_VEL
LIN {X 0,Y 404.115,Z 219.144,A -85,B 0,C 180,E1 -10778.579,E2 -10778.579} C_VEL
LIN {X 0,Y 404.185,Z 219.139,A -85,B 0,C 180,E1 -10781.761,E2 -10781.761} C_VEL
LIN {X 0,Y 404.183,Z 219.13,A -85,B 0,C 180,E1 -10784.881,E2 -10784.881} C_VEL
LIN {X 0,Y 404.229,Z 219.128,A -85,B 0,C 180,E1 -10787.958,E2 -10787.958} C_VEL
LIN {X 0,Y 404.381,Z 219.11,A -85,B 0,C 180,E1 -10792.127,E2 -10792.127} C_VEL
LIN {X 0,Y 404.399,Z 219.105,A -85,B 0,C 180,E1 -10794.015,E2 -10794.015} C_VEL
LIN {X 0,Y 404.449,Z 219.096,A -85,B 0,C 180,E1 -10798.008,E2 -10798.008} C_VEL
LIN {X 0,Y 404.58,Z 219.086,A -85,B 0,C 180,E1 -10800,E2 -10800} C_VEL
LIN {X 0,Y 404.384,Z 219.108,A -85,B 0,C 180,E1 -10802.989,E2 -10802.989} C_VEL
LIN {X 0,Y 404.353,Z 219.113,A -85,B 0,C 180,E1 -10806.988,E2 -10806.988} C_VEL
LIN {X 0,Y 404.232,Z 219.13,A -85,B 0,C 180,E1 -10811.025,E2 -10811.025} C_VEL
LIN {X 0,Y 404.183,Z 219.134,A -85,B 0,C 180,E1 -10814.089,E2 -10814.089} C_VEL
LIN {X 0,Y 404.182,Z 219.134,A -85,B 0,C 180,E1 -10817.193,E2 -10817.193} C_VEL
LIN {X 0,Y 404.132,Z 219.144,A -85,B 0,C 180,E1 -10820.353,E2 -10820.353} C_VEL
LIN {X 0,Y 404.133,Z 219.142,A -85,B 0,C 180,E1 -10823.577,E2 -10823.577} C_VEL
LIN {X 0,Y 404.11,Z 219.149,A -85,B 0,C 180,E1 -10826.883,E2 -10826.883} C_VEL
LIN {X 0,Y 404.123,Z 219.141,A -85,B 0,C 180,E1 -10830.287,E2 -10830.287} C_VEL
LIN {X 0,Y 404.12,Z 219.139,A -85,B 0,C 180,E1 -10833.815,E2 -10833.815} C_VEL
LIN {X 0,Y 404.118,Z 219.138,A -85,B 0,C 180,E1 -10836.876,E2 -10836.876} C_VEL
LIN {X 0,Y 404.135,Z 219.136,A -85,B 0,C 180,E1 -10840.082,E2 -10840.082} C_VEL
LIN {X 0,Y 404.139,Z 219.141,A -85,B 0,C 180,E1 -10843.085,E2 -10843.085} C_VEL
LIN {X 0,Y 404.136,Z 219.143,A -85,B 0,C 180,E1 -10845.927,E2 -10845.927} C_VEL
LIN {X 0,Y 404.098,Z 219.143,A -85,B 0,C 180,E1 -10848.635,E2 -10848.635} C_VEL
LIN {X 0,Y 404.133,Z 219.14,A -85,B 0,C 180,E1 -10851.496,E2 -10851.496} C_VEL
LIN {X 0,Y 404.179,Z 219.136,A -85,B 0,C 180,E1 -10854.985,E2 -10854.985} C_VEL
LIN {X 0,Y 404.138,Z 219.145,A -85,B 0,C 180,E1 -10858.555,E2 -10858.555} C_VEL
LIN {X 0,Y 404.173,Z 219.179,A -85,B 0,C 180,E1 -10860.568,E2 -10860.568} C_VEL
LIN {X 0,Y 406.611,Z 229.871,A -85,B 0,C 180,E1 -10863.019,E2 -10863.019} C_VEL
LIN {X 0,Y 408.085,Z 237.85,A -85,B 0,C 180,E1 -10864.771,E2 -10864.771} C_VEL
LIN {X 0,Y 407.071,Z 251.147,A -85,B 0,C 180,E1 -10867.41,E2 -10867.41} C_VEL
LIN {X 0,Y 406.233,Z 263.002,A -85,B 0,C 180,E1 -10869.734,E2 -10869.734} C_VEL
LIN {X 0,Y 410.621,Z 288.085,A -85,B 0,C 180,E1 -10870.463,E2 -10870.463} C_VEL
LIN {X 0,Y 411.228,Z 294.801,A -85,B 0,C 180,E1 -10870.622,E2 -10870.622} C_VEL
LIN {X 0,Y 410.197,Z 371.624,A -85,B 0,C 180,E1 -10872.008,E2 -10872.008} C_VEL
LIN {X 0,Y 409.589,Z 384.82,A -85,B 0,C 180,E1 -10872.429,E2 -10872.429} C_VEL
LIN {X 0,Y 408.784,Z 396.996,A -85,B 0,C 180,E1 -10873.006,E2 -10873.006} C_VEL
LIN {X 0,Y 407.896,Z 408.47,A -85,B 0,C 180,E1 -10873.74,E2 -10873.74} C_VEL
LIN {X 0,Y 406.964,Z 420.257,A -85,B 0,C 180,E1 -10874.73,E2 -10874.73} C_VEL
LIN {X 0,Y 406.065,Z 429.991,A -85,B 0,C 180,E1 -10875.749,E2 -10875.749} C_VEL
LIN {X 0,Y 405.282,Z 439.486,A -85,B 0,C 180,E1 -10876.971,E2 -10876.971} C_VEL
LIN {X 0,Y 404.533,Z 447.483,A -85,B 0,C 180,E1 -10878.22,E2 -10878.22} C_VEL
LIN {X 0,Y 403.87,Z 455.352,A -85,B 0,C 180,E1 -10879.724,E2 -10879.724} C_VEL
LIN {X 0,Y 403.32,Z 462.57,A -85,B 0,C 180,E1 -10881.481,E2 -10881.481} C_VEL
LIN {X 0,Y 403.075,Z 467.417,A -85,B 0,C 180,E1 -10882.988,E2 -10882.988} C_VEL
LIN {X 0,Y 402.893,Z 471.154,A -85,B 0,C 180,E1 -10884.493,E2 -10884.493} C_VEL
LIN {X 0,Y 402.855,Z 473.883,A -85,B 0,C 180,E1 -10885.997,E2 -10885.997} C_VEL
LIN {X 0,Y 402.946,Z 476.083,A -85,B 0,C 180,E1 -10887.999,E2 -10887.999} C_VEL
LIN {X 0,Y 402.905,Z 476.549,A -85,B 0,C 180,E1 -10888.999,E2 -10888.999} C_VEL
LIN {X 0,Y 402.898,Z 476.614,A -85,B 0,C 180,E1 -10889.998,E2 -10889.998} C_VEL
LIN {X 0,Y 402.95,Z 475.584,A -85,B 0,C 180,E1 -10891.997,E2 -10891.997} C_VEL
LIN {X 0,Y 402.899,Z 474.436,A -85,B 0,C 180,E1 -10892.998,E2 -10892.998} C_VEL
LIN {X 0,Y 402.863,Z 472.855,A -85,B 0,C 180,E1 -10893.999,E2 -10893.999} C_VEL
LIN {X 0,Y 402.922,Z 469.676,A -85,B 0,C 180,E1 -10895.503,E2 -10895.503} C_VEL
LIN {X 0,Y 403.072,Z 465.421,A -85,B 0,C 180,E1 -10897.008,E2 -10897.008} C_VEL
LIN {X 0,Y 403.326,Z 458.942,A -85,B 0,C 180,E1 -10898.767,E2 -10898.767} C_VEL
LIN {X 0,Y 403.688,Z 451.852,A -85,B 0,C 180,E1 -10900.276,E2 -10900.276} C_VEL
LIN {X 0,Y 404.334,Z 442.974,A -85,B 0,C 180,E1 -10901.782,E2 -10901.782} C_VEL
LIN {X 0,Y 404.963,Z 433.868,A -85,B 0,C 180,E1 -10903.036,E2 -10903.036} C_VEL
LIN {X 0,Y 405.684,Z 423.837,A -85,B 0,C 180,E1 -10904.161,E2 -10904.161} C_VEL
LIN {X 0,Y 406.333,Z 412.662,A -85,B 0,C 180,E1 -10905.162,E2 -10905.162} C_VEL
LIN {X 0,Y 407.127,Z 400.145,A -85,B 0,C 180,E1 -10906.03,E2 -10906.03} C_VEL
LIN {X 0,Y 407.808,Z 387.459,A -85,B 0,C 180,E1 -10906.678,E2 -10906.678} C_VEL
LIN {X 0,Y 408.347,Z 373.968,A -85,B 0,C 180,E1 -10907.138,E2 -10907.138} C_VEL
LIN {X 0,Y 408.78,Z 345.758,A -85,B 0,C 180,E1 -10907.668,E2 -10907.668} C_VEL
LIN {X 0,Y 409.22,Z 291.711,A -85,B 0,C 180,E1 -10908.619,E2 -10908.619} C_VEL
LIN {X 0,Y 405.348,Z 263.438,A -85,B 0,C 180,E1 -10909.296,E2 -10909.296} C_VEL
LIN {X 0,Y 406.495,Z 244.678,A -85,B 0,C 180,E1 -10912.888,E2 -10912.888} C_VEL
LIN {X 0,Y 407.03,Z 233.682,A -85,B 0,C 180,E1 -10915.021,E2 -10915.021} C_VEL
LIN {X 0,Y 404.647,Z 221.116,A -85,B 0,C 180,E1 -10917.652,E2 -10917.652} C_VEL
LIN {X 0,Y 404.244,Z 219.134,A -85,B 0,C 180,E1 -10918.132,E2 -10918.132} C_VEL
LIN {X 0,Y 404.122,Z 219.149,A -85,B 0,C 180,E1 -10921.554,E2 -10921.554} C_VEL
LIN {X 0,Y 404.165,Z 219.136,A -85,B 0,C 180,E1 -10925.012,E2 -10925.012} C_VEL
LIN {X 0,Y 404.13,Z 219.141,A -85,B 0,C 180,E1 -10928.753,E2 -10928.753} C_VEL
LIN {X 0,Y 404.096,Z 219.149,A -85,B 0,C 180,E1 -10931.595,E2 -10931.595} C_VEL
LIN {X 0,Y 404.121,Z 219.143,A -85,B 0,C 180,E1 -10934.518,E2 -10934.518} C_VEL
LIN {X 0,Y 404.174,Z 219.137,A -85,B 0,C 180,E1 -10937.3,E2 -10937.3} C_VEL
LIN {X 0,Y 404.136,Z 219.145,A -85,B 0,C 180,E1 -10939.951,E2 -10939.951} C_VEL
LIN {X 0,Y 404.104,Z 219.145,A -85,B 0,C 180,E1 -10943.121,E2 -10943.121} C_VEL
LIN {X 0,Y 404.106,Z 219.145,A -85,B 0,C 180,E1 -10946.184,E2 -10946.184} C_VEL
LIN {X 0,Y 404.111,Z 219.149,A -85,B 0,C 180,E1 -10949.712,E2 -10949.712} C_VEL
LIN {X 0,Y 404.152,Z 219.141,A -85,B 0,C 180,E1 -10953.12,E2 -10953.12} C_VEL
LIN {X 0,Y 404.139,Z 219.14,A -85,B 0,C 180,E1 -10956.424,E2 -10956.424} C_VEL
LIN {X 0,Y 404.181,Z 219.137,A -85,B 0,C 180,E1 -10959.858,E2 -10959.858} C_VEL
LIN {X 0,Y 404.169,Z 219.139,A -85,B 0,C 180,E1 -10962.99,E2 -10962.99} C_VEL
LIN {X 0,Y 404.217,Z 219.132,A -85,B 0,C 180,E1 -10966.787,E2 -10966.787} C_VEL
LIN {X 0,Y 404.223,Z 219.13,A -85,B 0,C 180,E1 -10969.987,E2 -10969.987} C_VEL
LIN {X 0,Y 404.373,Z 219.116,A -85,B 0,C 180,E1 -10973.012,E2 -10973.012} C_VEL
LIN {X 0,Y 404.237,Z 219.133,A -85,B 0,C 180,E1 -10975.013,E2 -10975.013} C_VEL
LIN {X 0,Y 404.428,Z 219.104,A -85,B 0,C 180,E1 -10978.008,E2 -10978.008} C_VEL
LIN {X 0,Y 404.556,Z 219.088,A -85,B 0,C 180,E1 -10980,E2 -10980} C_VEL
LIN {X 0,Y 404.362,Z 219.119,A -85,B 0,C 180,E1 -10982.989,E2 -10982.989} C_VEL
LIN {X 0,Y 404.35,Z 219.12,A -85,B 0,C 180,E1 -10986.988,E2 -10986.988} C_VEL
LIN {X 0,Y 404.211,Z 219.131,A -85,B 0,C 180,E1 -10990.013,E2 -10990.013} C_VEL
LIN {X 0,Y 404.217,Z 219.133,A -85,B 0,C 180,E1 -10993.213,E2 -10993.213} C_VEL
LIN {X 0,Y 404.169,Z 219.14,A -85,B 0,C 180,E1 -10997.01,E2 -10997.01} C_VEL
LIN {X 0,Y 404.108,Z 219.147,A -85,B 0,C 180,E1 -11000.355,E2 -11000.355} C_VEL
LIN {X 0,Y 404.118,Z 219.142,A -85,B 0,C 180,E1 -11003.578,E2 -11003.578} C_VEL
LIN {X 0,Y 404.14,Z 219.14,A -85,B 0,C 180,E1 -11005.77,E2 -11005.77} C_VEL
LIN {X 0,Y 404.155,Z 219.139,A -85,B 0,C 180,E1 -11008.003,E2 -11008.003} C_VEL
LIN {X 0,Y 404.101,Z 219.144,A -85,B 0,C 180,E1 -11011.562,E2 -11011.562} C_VEL
LIN {X 0,Y 404.147,Z 219.14,A -85,B 0,C 180,E1 -11015.02,E2 -11015.02} C_VEL
LIN {X 0,Y 404.126,Z 219.144,A -85,B 0,C 180,E1 -11018.761,E2 -11018.761} C_VEL
LIN {X 0,Y 404.158,Z 219.138,A -85,B 0,C 180,E1 -11021.614,E2 -11021.614} C_VEL
LIN {X 0,Y 404.154,Z 219.142,A -85,B 0,C 180,E1 -11024.532,E2 -11024.532} C_VEL
LIN {X 0,Y 404.11,Z 219.143,A -85,B 0,C 180,E1 -11027.3,E2 -11027.3} C_VEL
LIN {X 0,Y 404.146,Z 219.143,A -85,B 0,C 180,E1 -11029.96,E2 -11029.96} C_VEL
LIN {X 0,Y 404.116,Z 219.143,A -85,B 0,C 180,E1 -11033.13,E2 -11033.13} C_VEL
LIN {X 0,Y 404.127,Z 219.147,A -85,B 0,C 180,E1 -11036.192,E2 -11036.192} C_VEL
LIN {X 0,Y 404.131,Z 219.145,A -85,B 0,C 180,E1 -11039.719,E2 -11039.719} C_VEL
LIN {X 0,Y 404.183,Z 219.134,A -85,B 0,C 180,E1 -11043.127,E2 -11043.127} C_VEL
LIN {X 0,Y 404.164,Z 219.138,A -85,B 0,C 180,E1 -11045.338,E2 -11045.338} C_VEL
LIN {X 0,Y 404.131,Z 219.141,A -85,B 0,C 180,E1 -11048.584,E2 -11048.584} C_VEL
LIN {X 0,Y 404.199,Z 219.139,A -85,B 0,C 180,E1 -11051.765,E2 -11051.765} C_VEL
LIN {X 0,Y 404.202,Z 219.132,A -85,B 0,C 180,E1 -11054.885,E2 -11054.885} C_VEL
LIN {X 0,Y 404.254,Z 219.132,A -85,B 0,C 180,E1 -11057.962,E2 -11057.962} C_VEL
LIN {X 0,Y 404.26,Z 219.22,A -85,B 0,C 180,E1 -11059.612,E2 -11059.612} C_VEL
LIN {X 0,Y 405.808,Z 228.029,A -85,B 0,C 180,E1 -11061.681,E2 -11061.681} C_VEL
LIN {X 0,Y 405.828,Z 228.628,A -85,B 0,C 180,E1 -11061.815,E2 -11061.815} C_VEL
LIN {X 0,Y 409.748,Z 249.841,A -85,B 0,C 180,E1 -11062.364,E2 -11062.364} C_VEL
LIN {X 0,Y 408.568,Z 336.162,A -85,B 0,C 180,E1 -11063.893,E2 -11063.893} C_VEL
LIN {X 0,Y 408.148,Z 349.979,A -85,B 0,C 180,E1 -11064.351,E2 -11064.351} C_VEL
LIN {X 0,Y 407.721,Z 361.781,A -85,B 0,C 180,E1 -11064.934,E2 -11064.934} C_VEL
LIN {X 0,Y 407.273,Z 372.956,A -85,B 0,C 180,E1 -11065.673,E2 -11065.673} C_VEL
LIN {X 0,Y 406.439,Z 384.565,A -85,B 0,C 180,E1 -11066.657,E2 -11066.657} C_VEL
LIN {X 0,Y 405.735,Z 394.97,A -85,B 0,C 180,E1 -11067.768,E2 -11067.768} C_VEL
LIN {X 0,Y 405.085,Z 404.357,A -85,B 0,C 180,E1 -11069.008,E2 -11069.008} C_VEL
LIN {X 0,Y 404.931,Z 406.409,A -85,B 0,C 180,E1 -11069.322,E2 -11069.322} C_VEL
LIN {X 0,Y 404.027,Z 410.337,A -85,B 0,C 180,E1 -11069.936,E2 -11069.936} C_VEL
LIN {X 0,Y 400.693,Z 416.316,A -85,B 0,C 180,E1 -11070.959,E2 -11070.959} C_VEL
LIN {X 0,Y 397.42,Z 421.731,A -85,B 0,C 180,E1 -11072.061,E2 -11072.061} C_VEL
LIN {X 0,Y 396.625,Z 424.64,A -85,B 0,C 180,E1 -11072.791,E2 -11072.791} C_VEL
LIN {X 0,Y 396.4,Z 428.999,A -85,B 0,C 180,E1 -11074.068,E2 -11074.068} C_VEL
LIN {X 0,Y 396.158,Z 433.144,A -85,B 0,C 180,E1 -11075.601,E2 -11075.601} C_VEL
LIN {X 0,Y 395.967,Z 436.241,A -85,B 0,C 180,E1 -11077.138,E2 -11077.138} C_VEL
LIN {X 0,Y 395.856,Z 437.786,A -85,B 0,C 180,E1 -11078.167,E2 -11078.167} C_VEL
LIN {X 0,Y 395.775,Z 438.876,A -85,B 0,C 180,E1 -11079.197,E2 -11079.197} C_VEL
LIN {X 0,Y 395.79,Z 439.862,A -85,B 0,C 180,E1 -11081.265,E2 -11081.265} C_VEL
LIN {X 0,Y 395.844,Z 439.703,A -85,B 0,C 180,E1 -11082.446,E2 -11082.446} C_VEL
LIN {X 0,Y 395.904,Z 438.277,A -85,B 0,C 180,E1 -11084.391,E2 -11084.391} C_VEL
LIN {X 0,Y 396.047,Z 436.926,A -85,B 0,C 180,E1 -11085.438,E2 -11085.438} C_VEL
LIN {X 0,Y 396.34,Z 434.555,A -85,B 0,C 180,E1 -11086.755,E2 -11086.755} C_VEL
LIN {X 0,Y 396.721,Z 430.048,A -85,B 0,C 180,E1 -11088.595,E2 -11088.595} C_VEL
LIN {X 0,Y 397.317,Z 424.14,A -85,B 0,C 180,E1 -11090.363,E2 -11090.363} C_VEL
LIN {X 0,Y 398.054,Z 416.937,A -85,B 0,C 180,E1 -11092.036,E2 -11092.036} C_VEL
LIN {X 0,Y 398.961,Z 408.875,A -85,B 0,C 180,E1 -11093.527,E2 -11093.527} C_VEL
LIN {X 0,Y 399.862,Z 399.272,A -85,B 0,C 180,E1 -11094.949,E2 -11094.949} C_VEL
LIN {X 0,Y 400.847,Z 388.809,A -85,B 0,C 180,E1 -11096.193,E2 -11096.193} C_VEL
LIN {X 0,Y 401.821,Z 378.286,A -85,B 0,C 180,E1 -11097.189,E2 -11097.189} C_VEL
LIN {X 0,Y 402.558,Z 366.759,A -85,B 0,C 180,E1 -11098.052,E2 -11098.052} C_VEL
LIN {X 0,Y 403.203,Z 355.145,A -85,B 0,C 180,E1 -11098.712,E2 -11098.712} C_VEL
LIN {X 0,Y 403.762,Z 341.965,A -85,B 0,C 180,E1 -11099.242,E2 -11099.242} C_VEL
LIN {X 0,Y 404.085,Z 327.267,A -85,B 0,C 180,E1 -11099.585,E2 -11099.585} C_VEL
LIN {X 0,Y 405.22,Z 249.976,A -85,B 0,C 180,E1 -11100.98,E2 -11100.98} C_VEL
LIN {X 0,Y 401.516,Z 235.467,A -85,B 0,C 180,E1 -11101.488,E2 -11101.488} C_VEL
LIN {X 0,Y 399.164,Z 229.267,A -85,B 0,C 180,E1 -11101.773,E2 -11101.773} C_VEL
LIN {X 0,Y 397.133,Z 220.017,A -85,B 0,C 180,E1 -11104.171,E2 -11104.171} C_VEL
LIN {X 0,Y 397.094,Z 220.024,A -85,B 0,C 180,E1 -11107.208,E2 -11107.208} C_VEL
LIN {X 0,Y 397.113,Z 220.017,A -85,B 0,C 180,E1 -11110.447,E2 -11110.447} C_VEL
LIN {X 0,Y 397.094,Z 220.017,A -85,B 0,C 180,E1 -11113.647,E2 -11113.647} C_VEL
LIN {X 0,Y 397.147,Z 220.016,A -85,B 0,C 180,E1 -11116.511,E2 -11116.511} C_VEL
LIN {X 0,Y 397.11,Z 220.02,A -85,B 0,C 180,E1 -11119.549,E2 -11119.549} C_VEL
LIN {X 0,Y 397.084,Z 220.018,A -85,B 0,C 180,E1 -11122.789,E2 -11122.789} C_VEL
LIN {X 0,Y 397.102,Z 220.02,A -85,B 0,C 180,E1 -11126.281,E2 -11126.281} C_VEL
LIN {X 0,Y 397.095,Z 220.023,A -85,B 0,C 180,E1 -11130.132,E2 -11130.132} C_VEL
LIN {X 0,Y 397.176,Z 220.004,A -85,B 0,C 180,E1 -11132.608,E2 -11132.608} C_VEL
LIN {X 0,Y 397.108,Z 220.014,A -85,B 0,C 180,E1 -11135.98,E2 -11135.98} C_VEL
LIN {X 0,Y 397.095,Z 220.017,A -85,B 0,C 180,E1 -11139.712,E2 -11139.712} C_VEL
LIN {X 0,Y 397.161,Z 220.011,A -85,B 0,C 180,E1 -11142.843,E2 -11142.843} C_VEL
LIN {X 0,Y 397.206,Z 220.005,A -85,B 0,C 180,E1 -11146.702,E2 -11146.702} C_VEL
LIN {X 0,Y 397.191,Z 220.008,A -85,B 0,C 180,E1 -11149.808,E2 -11149.808} C_VEL
LIN {X 0,Y 397.333,Z 219.99,A -85,B 0,C 180,E1 -11152.887,E2 -11152.887} C_VEL
LIN {X 0,Y 397.227,Z 220.001,A -85,B 0,C 180,E1 -11154.925,E2 -11154.925} C_VEL
LIN {X 0,Y 397.418,Z 219.971,A -85,B 0,C 180,E1 -11157.973,E2 -11157.973} C_VEL
LIN {X 0,Y 397.55,Z 219.961,A -85,B 0,C 180,E1 -11160,E2 -11160} C_VEL
LIN {X 0,Y 397.343,Z 219.985,A -85,B 0,C 180,E1 -11163.042,E2 -11163.042} C_VEL
LIN {X 0,Y 397.301,Z 219.99,A -85,B 0,C 180,E1 -11167.113,E2 -11167.113} C_VEL
LIN {X 0,Y 397.193,Z 220.006,A -85,B 0,C 180,E1 -11170.192,E2 -11170.192} C_VEL
LIN {X 0,Y 397.203,Z 220.006,A -85,B 0,C 180,E1 -11173.322,E2 -11173.322} C_VEL
LIN {X 0,Y 397.162,Z 220.008,A -85,B 0,C 180,E1 -11177.157,E2 -11177.157} C_VEL
LIN {X 0,Y 397.075,Z 220.02,A -85,B 0,C 180,E1 -11180.731,E2 -11180.731} C_VEL
LIN {X 0,Y 397.095,Z 220.019,A -85,B 0,C 180,E1 -11184.021,E2 -11184.021} C_VEL
LIN {X 0,Y 397.071,Z 220.022,A -85,B 0,C 180,E1 -11187.758,E2 -11187.758} C_VEL
LIN {X 0,Y 397.057,Z 220.027,A -85,B 0,C 180,E1 -11190.884,E2 -11190.884} C_VEL
LIN {X 0,Y 397.1,Z 220.019,A -85,B 0,C 180,E1 -11194.496,E2 -11194.496} C_VEL
LIN {X 0,Y 397.082,Z 220.006,A -85,B 0,C 180,E1 -11198.277,E2 -11198.277} C_VEL
LIN {X 0,Y 397.073,Z 220.023,A -85,B 0,C 180,E1 -11200.911,E2 -11200.911} C_VEL
LIN {X 0,Y 397.089,Z 220.02,A -85,B 0,C 180,E1 -11203.65,E2 -11203.65} C_VEL
LIN {X 0,Y 397.09,Z 220.022,A -85,B 0,C 180,E1 -11206.523,E2 -11206.523} C_VEL
LIN {X 0,Y 397.078,Z 220.023,A -85,B 0,C 180,E1 -11210.421,E2 -11210.421} C_VEL
LIN {X 0,Y 397.09,Z 220.022,A -85,B 0,C 180,E1 -11213.006,E2 -11213.006} C_VEL
LIN {X 0,Y 397.114,Z 220.019,A -85,B 0,C 180,E1 -11216.283,E2 -11216.283} C_VEL
LIN {X 0,Y 397.129,Z 220.051,A -85,B 0,C 180,E1 -11220.187,E2 -11220.187} C_VEL
LIN {X 0,Y 399.921,Z 232.319,A -85,B 0,C 180,E1 -11223.056,E2 -11223.056} C_VEL
LIN {X 0,Y 401.191,Z 239.15,A -85,B 0,C 180,E1 -11224.585,E2 -11224.585} C_VEL
LIN {X 0,Y 400.619,Z 247.117,A -85,B 0,C 180,E1 -11226.204,E2 -11226.204} C_VEL
LIN {X 0,Y 399.364,Z 262.669,A -85,B 0,C 180,E1 -11229.313,E2 -11229.313} C_VEL
LIN {X 0,Y 403.753,Z 287.022,A -85,B 0,C 180,E1 -11230.045,E2 -11230.045} C_VEL
LIN {X 0,Y 404.657,Z 294.908,A -85,B 0,C 180,E1 -11230.248,E2 -11230.248} C_VEL
LIN {X 0,Y 403.538,Z 372.082,A -85,B 0,C 180,E1 -11231.669,E2 -11231.669} C_VEL
LIN {X 0,Y 402.874,Z 385.725,A -85,B 0,C 180,E1 -11232.126,E2 -11232.126} C_VEL
LIN {X 0,Y 402.03,Z 397.577,A -85,B 0,C 180,E1 -11232.711,E2 -11232.711} C_VEL
LIN {X 0,Y 401.117,Z 408.813,A -85,B 0,C 180,E1 -11233.458,E2 -11233.458} C_VEL
LIN {X 0,Y 400.11,Z 420.439,A -85,B 0,C 180,E1 -11234.462,E2 -11234.462} C_VEL
LIN {X 0,Y 399.09,Z 430.9,A -85,B 0,C 180,E1 -11235.594,E2 -11235.594} C_VEL
LIN {X 0,Y 398.348,Z 439.505,A -85,B 0,C 180,E1 -11236.74,E2 -11236.74} C_VEL
LIN {X 0,Y 397.578,Z 447.442,A -85,B 0,C 180,E1 -11238.011,E2 -11238.011} C_VEL
LIN {X 0,Y 396.854,Z 455.237,A -85,B 0,C 180,E1 -11239.541,E2 -11239.541} C_VEL
LIN {X 0,Y 396.286,Z 462.411,A -85,B 0,C 180,E1 -11241.329,E2 -11241.329} C_VEL
LIN {X 0,Y 396.002,Z 467.222,A -85,B 0,C 180,E1 -11242.862,E2 -11242.862} C_VEL
LIN {X 0,Y 395.816,Z 470.534,A -85,B 0,C 180,E1 -11244.209,E2 -11244.209} C_VEL
LIN {X 0,Y 395.777,Z 473.622,A -85,B 0,C 180,E1 -11245.925,E2 -11245.925} C_VEL
LIN {X 0,Y 395.856,Z 475.787,A -85,B 0,C 180,E1 -11247.963,E2 -11247.963} C_VEL
LIN {X 0,Y 395.832,Z 476.23,A -85,B 0,C 180,E1 -11248.981,E2 -11248.981} C_VEL
LIN {X 0,Y 395.823,Z 476.28,A -85,B 0,C 180,E1 -11249.998,E2 -11249.998} C_VEL
LIN {X 0,Y 395.88,Z 475.219,A -85,B 0,C 180,E1 -11252.033,E2 -11252.033} C_VEL
LIN {X 0,Y 395.8,Z 474.041,A -85,B 0,C 180,E1 -11253.051,E2 -11253.051} C_VEL
LIN {X 0,Y 395.827,Z 471.509,A -85,B 0,C 180,E1 -11254.58,E2 -11254.58} C_VEL
LIN {X 0,Y 395.928,Z 466.651,A -85,B 0,C 180,E1 -11256.572,E2 -11256.572} C_VEL
LIN {X 0,Y 396.121,Z 461.434,A -85,B 0,C 180,E1 -11258.157,E2 -11258.157} C_VEL
LIN {X 0,Y 396.435,Z 455.048,A -85,B 0,C 180,E1 -11259.693,E2 -11259.693} C_VEL
LIN {X 0,Y 396.966,Z 447.039,A -85,B 0,C 180,E1 -11261.227,E2 -11261.227} C_VEL
LIN {X 0,Y 397.568,Z 438.875,A -85,B 0,C 180,E1 -11262.503,E2 -11262.503} C_VEL
LIN {X 0,Y 398.264,Z 428.783,A -85,B 0,C 180,E1 -11263.793,E2 -11263.793} C_VEL
LIN {X 0,Y 399.056,Z 417.692,A -85,B 0,C 180,E1 -11264.922,E2 -11264.922} C_VEL
LIN {X 0,Y 399.798,Z 406.695,A -85,B 0,C 180,E1 -11265.808,E2 -11265.808} C_VEL
LIN {X 0,Y 400.555,Z 394.544,A -85,B 0,C 180,E1 -11266.562,E2 -11266.562} C_VEL
LIN {X 0,Y 401.201,Z 382.035,A -85,B 0,C 180,E1 -11267.125,E2 -11267.125} C_VEL
LIN {X 0,Y 401.646,Z 368.992,A -85,B 0,C 180,E1 -11267.499,E2 -11267.499} C_VEL
LIN {X 0,Y 402.466,Z 293.403,A -85,B 0,C 180,E1 -11268.854,E2 -11268.854} C_VEL
LIN {X 0,Y 398.384,Z 263.17,A -85,B 0,C 180,E1 -11269.58,E2 -11269.58} C_VEL
LIN {X 0,Y 399.603,Z 244.056,A -85,B 0,C 180,E1 -11273.306,E2 -11273.306} C_VEL
LIN {X 0,Y 400.094,Z 235.815,A -85,B 0,C 180,E1 -11274.93,E2 -11274.93} C_VEL
LIN {X 0,Y 398.66,Z 227.371,A -85,B 0,C 180,E1 -11276.709,E2 -11276.709} C_VEL
LIN {X 0,Y 397.176,Z 220.014,A -85,B 0,C 180,E1 -11278.34,E2 -11278.34} C_VEL
LIN {X 0,Y 397.061,Z 220.029,A -85,B 0,C 180,E1 -11282.067,E2 -11282.067} C_VEL
LIN {X 0,Y 397.099,Z 220.019,A -85,B 0,C 180,E1 -11285.499,E2 -11285.499} C_VEL
LIN {X 0,Y 397.106,Z 220.016,A -85,B 0,C 180,E1 -11288.857,E2 -11288.857} C_VEL
LIN {X 0,Y 397.041,Z 220.027,A -85,B 0,C 180,E1 -11292.263,E2 -11292.263} C_VEL
LIN {X 0,Y 397.081,Z 220.019,A -85,B 0,C 180,E1 -11295.061,E2 -11295.061} C_VEL
LIN {X 0,Y 397.124,Z 220.018,A -85,B 0,C 180,E1 -11298.003,E2 -11298.003} C_VEL
LIN {X 0,Y 397.075,Z 220.027,A -85,B 0,C 180,E1 -11301.722,E2 -11301.722} C_VEL
LIN {X 0,Y 397.087,Z 220.023,A -85,B 0,C 180,E1 -11305.503,E2 -11305.503} C_VEL
LIN {X 0,Y 397.042,Z 220.026,A -85,B 0,C 180,E1 -11309.114,E2 -11309.114} C_VEL
LIN {X 0,Y 397.152,Z 220.01,A -85,B 0,C 180,E1 -11312.607,E2 -11312.607} C_VEL
LIN {X 0,Y 397.096,Z 220.019,A -85,B 0,C 180,E1 -11315.979,E2 -11315.979} C_VEL
LIN {X 0,Y 397.113,Z 220.02,A -85,B 0,C 180,E1 -11319.271,E2 -11319.271} C_VEL
LIN {X 0,Y 397.135,Z 220.014,A -85,B 0,C 180,E1 -11322.842,E2 -11322.842} C_VEL
LIN {X 0,Y 397.133,Z 220.015,A -85,B 0,C 180,E1 -11325.655,E2 -11325.655} C_VEL
LIN {X 0,Y 397.16,Z 220.011,A -85,B 0,C 180,E1 -11328.776,E2 -11328.776} C_VEL
LIN {X 0,Y 397.346,Z 219.986,A -85,B 0,C 180,E1 -11332.038,E2 -11332.038} C_VEL
LIN {X 0,Y 397.343,Z 219.987,A -85,B 0,C 180,E1 -11333.908,E2 -11333.908} C_VEL
LIN {X 0,Y 397.398,Z 219.98,A -85,B 0,C 180,E1 -11337.973,E2 -11337.973} C_VEL
LIN {X 0,Y 397.526,Z 219.964,A -85,B 0,C 180,E1 -11340,E2 -11340} C_VEL
LIN {X 0,Y 397.322,Z 219.996,A -85,B 0,C 180,E1 -11343.042,E2 -11343.042} C_VEL
LIN {X 0,Y 397.293,Z 219.993,A -85,B 0,C 180,E1 -11346.689,E2 -11346.689} C_VEL
LIN {X 0,Y 397.202,Z 220.008,A -85,B 0,C 180,E1 -11349.163,E2 -11349.163} C_VEL
LIN {X 0,Y 397.179,Z 220.008,A -85,B 0,C 180,E1 -11352.26,E2 -11352.26} C_VEL
LIN {X 0,Y 397.134,Z 220.013,A -85,B 0,C 180,E1 -11355.394,E2 -11355.394} C_VEL
LIN {X 0,Y 397.113,Z 220.02,A -85,B 0,C 180,E1 -11358.576,E2 -11358.576} C_VEL
LIN {X 0,Y 397.048,Z 220.023,A -85,B 0,C 180,E1 -11361.822,E2 -11361.822} C_VEL
LIN {X 0,Y 397.109,Z 220.016,A -85,B 0,C 180,E1 -11365.515,E2 -11365.515} C_VEL
LIN {X 0,Y 397.085,Z 220.026,A -85,B 0,C 180,E1 -11368.547,E2 -11368.547} C_VEL
LIN {X 0,Y 397.04,Z 220.027,A -85,B 0,C 180,E1 -11372.075,E2 -11372.075} C_VEL
LIN {X 0,Y 397.082,Z 220.019,A -85,B 0,C 180,E1 -11375.507,E2 -11375.507} C_VEL
LIN {X 0,Y 397.1,Z 220.018,A -85,B 0,C 180,E1 -11378.866,E2 -11378.866} C_VEL
LIN {X 0,Y 397.126,Z 220.02,A -85,B 0,C 180,E1 -11382.26,E2 -11382.26} C_VEL
LIN {X 0,Y 397.078,Z 220.02,A -85,B 0,C 180,E1 -11385.071,E2 -11385.071} C_VEL
LIN {X 0,Y 397.041,Z 220.029,A -85,B 0,C 180,E1 -11388.026,E2 -11388.026} C_VEL
LIN {X 0,Y 397.109,Z 220.015,A -85,B 0,C 180,E1 -11391.143,E2 -11391.143} C_VEL
LIN {X 0,Y 397.1,Z 220.019,A -85,B 0,C 180,E1 -11394.501,E2 -11394.501} C_VEL
LIN {X 0,Y 397.062,Z 220.027,A -85,B 0,C 180,E1 -11397.933,E2 -11397.933} C_VEL
LIN {X 0,Y 397.109,Z 220.017,A -85,B 0,C 180,E1 -11401.461,E2 -11401.461} C_VEL
LIN {X 0,Y 397.142,Z 220.013,A -85,B 0,C 180,E1 -11404.492,E2 -11404.492} C_VEL
LIN {X 0,Y 397.088,Z 220.021,A -85,B 0,C 180,E1 -11408.185,E2 -11408.185} C_VEL
LIN {X 0,Y 397.152,Z 220.013,A -85,B 0,C 180,E1 -11411.43,E2 -11411.43} C_VEL
LIN {X 0,Y 397.175,Z 220.007,A -85,B 0,C 180,E1 -11414.611,E2 -11414.611} C_VEL
LIN {X 0,Y 397.217,Z 220.009,A -85,B 0,C 180,E1 -11417.745,E2 -11417.745} C_VEL
LIN {X 0,Y 397.239,Z 220.149,A -85,B 0,C 180,E1 -11419.426,E2 -11419.426} C_VEL
LIN {X 0,Y 398.818,Z 228.937,A -85,B 0,C 180,E1 -11421.519,E2 -11421.519} C_VEL
LIN {X 0,Y 402.931,Z 250.358,A -85,B 0,C 180,E1 -11422.092,E2 -11422.092} C_VEL
LIN {X 0,Y 401.711,Z 336.042,A -85,B 0,C 180,E1 -11423.63,E2 -11423.63} C_VEL
LIN {X 0,Y 401.276,Z 349.27,A -85,B 0,C 180,E1 -11424.065,E2 -11424.065} C_VEL
LIN {X 0,Y 400.951,Z 360.191,A -85,B 0,C 180,E1 -11424.596,E2 -11424.596} C_VEL
LIN {X 0,Y 400.482,Z 371.809,A -85,B 0,C 180,E1 -11425.347,E2 -11425.347} C_VEL
LIN {X 0,Y 399.723,Z 382.472,A -85,B 0,C 180,E1 -11426.222,E2 -11426.222} C_VEL
LIN {X 0,Y 399.037,Z 392.265,A -85,B 0,C 180,E1 -11427.226,E2 -11427.226} C_VEL
LIN {X 0,Y 398.262,Z 402.182,A -85,B 0,C 180,E1 -11428.485,E2 -11428.485} C_VEL
LIN {X 0,Y 397.57,Z 411.78,A -85,B 0,C 180,E1 -11430.002,E2 -11430.002} C_VEL
LIN {X 0,Y 396.925,Z 419.459,A -85,B 0,C 180,E1 -11431.524,E2 -11431.524} C_VEL
LIN {X 0,Y 396.625,Z 424.64,A -85,B 0,C 180,E1 -11432.791,E2 -11432.791} C_VEL
LIN {X 0,Y 395.875,Z 427.388,A -85,B 0,C 180,E1 -11433.542,E2 -11433.542} C_VEL
LIN {X 0,Y 392.807,Z 431.317,A -85,B 0,C 180,E1 -11434.786,E2 -11434.786} C_VEL
LIN {X 0,Y 390.201,Z 434.018,A -85,B 0,C 180,E1 -11435.819,E2 -11435.819} C_VEL
LIN {X 0,Y 389.035,Z 435.736,A -85,B 0,C 180,E1 -11436.638,E2 -11436.638} C_VEL
LIN {X 0,Y 388.915,Z 436.206,A -85,B 0,C 180,E1 -11436.919,E2 -11436.919} C_VEL
LIN {X 0,Y 388.771,Z 438.287,A -85,B 0,C 180,E1 -11438.316,E2 -11438.316} C_VEL
LIN {X 0,Y 388.661,Z 439.963,A -85,B 0,C 180,E1 -11440.419,E2 -11440.419} C_VEL
LIN {X 0,Y 388.699,Z 440.215,A -85,B 0,C 180,E1 -11441.473,E2 -11441.473} C_VEL
LIN {X 0,Y 388.773,Z 440.028,A -85,B 0,C 180,E1 -11442.529,E2 -11442.529} C_VEL
LIN {X 0,Y 388.862,Z 438.443,A -85,B 0,C 180,E1 -11444.657,E2 -11444.657} C_VEL
LIN {X 0,Y 389.027,Z 437.028,A -85,B 0,C 180,E1 -11445.723,E2 -11445.723} C_VEL
LIN {X 0,Y 389.338,Z 434.154,A -85,B 0,C 180,E1 -11447.274,E2 -11447.274} C_VEL
LIN {X 0,Y 389.757,Z 429.938,A -85,B 0,C 180,E1 -11448.94,E2 -11448.94} C_VEL
LIN {X 0,Y 390.353,Z 424.518,A -85,B 0,C 180,E1 -11450.573,E2 -11450.573} C_VEL
LIN {X 0,Y 391.071,Z 417.811,A -85,B 0,C 180,E1 -11452.172,E2 -11452.172} C_VEL
LIN {X 0,Y 392.115,Z 409.229,A -85,B 0,C 180,E1 -11453.8,E2 -11453.8} C_VEL
LIN {X 0,Y 393.084,Z 399.47,A -85,B 0,C 180,E1 -11455.268,E2 -11455.268} C_VEL
LIN {X 0,Y 394.069,Z 389.47,A -85,B 0,C 180,E1 -11456.478,E2 -11456.478} C_VEL
LIN {X 0,Y 395.128,Z 378.406,A -85,B 0,C 180,E1 -11457.545,E2 -11457.545} C_VEL
LIN {X 0,Y 395.923,Z 366.822,A -85,B 0,C 180,E1 -11458.42,E2 -11458.42} C_VEL
LIN {X 0,Y 396.591,Z 355.122,A -85,B 0,C 180,E1 -11459.091,E2 -11459.091} C_VEL
LIN {X 0,Y 397.165,Z 341.856,A -85,B 0,C 180,E1 -11459.627,E2 -11459.627} C_VEL
LIN {X 0,Y 397.528,Z 326.429,A -85,B 0,C 180,E1 -11459.981,E2 -11459.981} C_VEL
LIN {X 0,Y 398.719,Z 251.264,A -85,B 0,C 180,E1 -11461.359,E2 -11461.359} C_VEL
LIN {X 0,Y 395.329,Z 237.975,A -85,B 0,C 180,E1 -11461.836,E2 -11461.836} C_VEL
LIN {X 0,Y 392.036,Z 229.656,A -85,B 0,C 180,E1 -11462.228,E2 -11462.228} C_VEL
LIN {X 0,Y 390.12,Z 220.892,A -85,B 0,C 180,E1 -11464.499,E2 -11464.499} C_VEL
LIN {X 0,Y 390.042,Z 220.904,A -85,B 0,C 180,E1 -11467.778,E2 -11467.778} C_VEL
LIN {X 0,Y 390.069,Z 220.896,A -85,B 0,C 180,E1 -11470.823,E2 -11470.823} C_VEL
LIN {X 0,Y 390.05,Z 220.893,A -85,B 0,C 180,E1 -11473.885,E2 -11473.885} C_VEL
LIN {X 0,Y 390.101,Z 220.892,A -85,B 0,C 180,E1 -11476.795,E2 -11476.795} C_VEL
LIN {X 0,Y 390.064,Z 220.897,A -85,B 0,C 180,E1 -11479.561,E2 -11479.561} C_VEL
LIN {X 0,Y 390.033,Z 220.897,A -85,B 0,C 180,E1 -11482.447,E2 -11482.447} C_VEL
LIN {X 0,Y 390.052,Z 220.897,A -85,B 0,C 180,E1 -11486.043,E2 -11486.043} C_VEL
LIN {X 0,Y 390.034,Z 220.9,A -85,B 0,C 180,E1 -11489.867,E2 -11489.867} C_VEL
LIN {X 0,Y 390.094,Z 220.887,A -85,B 0,C 180,E1 -11493.23,E2 -11493.23} C_VEL
LIN {X 0,Y 390.047,Z 220.891,A -85,B 0,C 180,E1 -11496.763,E2 -11496.763} C_VEL
LIN {X 0,Y 390.064,Z 220.89,A -85,B 0,C 180,E1 -11499.981,E2 -11499.981} C_VEL
LIN {X 0,Y 390.117,Z 220.891,A -85,B 0,C 180,E1 -11503.247,E2 -11503.247} C_VEL
LIN {X 0,Y 390.172,Z 220.881,A -85,B 0,C 180,E1 -11506.561,E2 -11506.561} C_VEL
LIN {X 0,Y 390.179,Z 220.879,A -85,B 0,C 180,E1 -11510.67,E2 -11510.67} C_VEL
LIN {X 0,Y 390.304,Z 220.862,A -85,B 0,C 180,E1 -11513.798,E2 -11513.798} C_VEL
LIN {X 0,Y 390.388,Z 220.847,A -85,B 0,C 180,E1 -11517.936,E2 -11517.936} C_VEL
LIN {X 0,Y 390.52,Z 220.837,A -85,B 0,C 180,E1 -11520,E2 -11520} C_VEL
LIN {X 0,Y 390.278,Z 220.865,A -85,B 0,C 180,E1 -11523.097,E2 -11523.097} C_VEL
LIN {X 0,Y 390.274,Z 220.867,A -85,B 0,C 180,E1 -11526.203,E2 -11526.203} C_VEL
LIN {X 0,Y 390.168,Z 220.884,A -85,B 0,C 180,E1 -11529.33,E2 -11529.33} C_VEL
LIN {X 0,Y 390.15,Z 220.879,A -85,B 0,C 180,E1 -11532.484,E2 -11532.484} C_VEL
LIN {X 0,Y 390.114,Z 220.886,A -85,B 0,C 180,E1 -11535.678,E2 -11535.678} C_VEL
LIN {X 0,Y 390.073,Z 220.898,A -85,B 0,C 180,E1 -11538.924,E2 -11538.924} C_VEL
LIN {X 0,Y 390.012,Z 220.897,A -85,B 0,C 180,E1 -11542.236,E2 -11542.236} C_VEL
LIN {X 0,Y 390.031,Z 220.892,A -85,B 0,C 180,E1 -11545.723,E2 -11545.723} C_VEL
LIN {X 0,Y 390.012,Z 220.897,A -85,B 0,C 180,E1 -11549.113,E2 -11549.113} C_VEL
LIN {X 0,Y 390.023,Z 220.898,A -85,B 0,C 180,E1 -11552.723,E2 -11552.723} C_VEL
LIN {X 0,Y 390.027,Z 220.9,A -85,B 0,C 180,E1 -11555.824,E2 -11555.824} C_VEL
LIN {X 0,Y 390.03,Z 220.887,A -85,B 0,C 180,E1 -11559.215,E2 -11559.215} C_VEL
LIN {X 0,Y 390.028,Z 220.901,A -85,B 0,C 180,E1 -11562.375,E2 -11562.375} C_VEL
LIN {X 0,Y 390.032,Z 220.897,A -85,B 0,C 180,E1 -11565.355,E2 -11565.355} C_VEL
LIN {X 0,Y 390.011,Z 220.896,A -85,B 0,C 180,E1 -11568.186,E2 -11568.186} C_VEL
LIN {X 0,Y 390.05,Z 220.896,A -85,B 0,C 180,E1 -11570.905,E2 -11570.905} C_VEL
LIN {X 0,Y 390.08,Z 220.891,A -85,B 0,C 180,E1 -11574.794,E2 -11574.794} C_VEL
LIN {X 0,Y 390.02,Z 220.904,A -85,B 0,C 180,E1 -11578.497,E2 -11578.497} C_VEL
LIN {X 0,Y 390.061,Z 220.992,A -85,B 0,C 180,E1 -11579.803,E2 -11579.803} C_VEL
LIN {X 0,Y 392.724,Z 232.48,A -85,B 0,C 180,E1 -11582.562,E2 -11582.562} C_VEL
LIN {X 0,Y 394.286,Z 240.453,A -85,B 0,C 180,E1 -11584.39,E2 -11584.39} C_VEL
LIN {X 0,Y 394.161,Z 244.093,A -85,B 0,C 180,E1 -11585.155,E2 -11585.155} C_VEL
LIN {X 0,Y 392.536,Z 262.32,A -85,B 0,C 180,E1 -11588.872,E2 -11588.872} C_VEL
LIN {X 0,Y 396.739,Z 285.141,A -85,B 0,C 180,E1 -11589.585,E2 -11589.585} C_VEL
LIN {X 0,Y 398.117,Z 295.305,A -85,B 0,C 180,E1 -11589.866,E2 -11589.866} C_VEL
LIN {X 0,Y 396.952,Z 371.461,A -85,B 0,C 180,E1 -11591.289,E2 -11591.289} C_VEL
LIN {X 0,Y 396.253,Z 385.168,A -85,B 0,C 180,E1 -11591.75,E2 -11591.75} C_VEL
LIN {X 0,Y 395.393,Z 397.077,A -85,B 0,C 180,E1 -11592.345,E2 -11592.345} C_VEL
LIN {X 0,Y 394.35,Z 409.155,A -85,B 0,C 180,E1 -11593.165,E2 -11593.165} C_VEL
LIN {X 0,Y 393.294,Z 420.654,A -85,B 0,C 180,E1 -11594.186,E2 -11594.186} C_VEL
LIN {X 0,Y 392.16,Z 431.62,A -85,B 0,C 180,E1 -11595.409,E2 -11595.409} C_VEL
LIN {X 0,Y 391.269,Z 441.22,A -85,B 0,C 180,E1 -11596.76,E2 -11596.76} C_VEL
LIN {X 0,Y 390.274,Z 450.154,A -85,B 0,C 180,E1 -11598.311,E2 -11598.311} C_VEL
LIN {X 0,Y 389.614,Z 457.371,A -85,B 0,C 180,E1 -11599.869,E2 -11599.869} C_VEL
LIN {X 0,Y 389.105,Z 463.978,A -85,B 0,C 180,E1 -11601.691,E2 -11601.691} C_VEL
LIN {X 0,Y 388.85,Z 468.369,A -85,B 0,C 180,E1 -11603.252,E2 -11603.252} C_VEL
LIN {X 0,Y 388.729,Z 471.699,A -85,B 0,C 180,E1 -11604.812,E2 -11604.812} C_VEL
LIN {X 0,Y 388.7,Z 473.364,A -85,B 0,C 180,E1 -11605.851,E2 -11605.851} C_VEL
LIN {X 0,Y 388.668,Z 474.628,A -85,B 0,C 180,E1 -11606.889,E2 -11606.889} C_VEL
LIN {X 0,Y 388.754,Z 475.487,A -85,B 0,C 180,E1 -11607.926,E2 -11607.926} C_VEL
LIN {X 0,Y 388.762,Z 475.91,A -85,B 0,C 180,E1 -11608.962,E2 -11608.962} C_VEL
LIN {X 0,Y 388.762,Z 475.595,A -85,B 0,C 180,E1 -11611.034,E2 -11611.034} C_VEL
LIN {X 0,Y 388.792,Z 474.846,A -85,B 0,C 180,E1 -11612.07,E2 -11612.07} C_VEL
LIN {X 0,Y 388.702,Z 473.643,A -85,B 0,C 180,E1 -11613.107,E2 -11613.107} C_VEL
LIN {X 0,Y 388.762,Z 471.08,A -85,B 0,C 180,E1 -11614.664,E2 -11614.664} C_VEL
LIN {X 0,Y 388.792,Z 467.482,A -85,B 0,C 180,E1 -11616.224,E2 -11616.224} C_VEL
LIN {X 0,Y 388.98,Z 462.762,A -85,B 0,C 180,E1 -11617.785,E2 -11617.785} C_VEL
LIN {X 0,Y 389.329,Z 455.639,A -85,B 0,C 180,E1 -11619.609,E2 -11619.609} C_VEL
LIN {X 0,Y 389.822,Z 447.909,A -85,B 0,C 180,E1 -11621.172,E2 -11621.172} C_VEL
LIN {X 0,Y 390.45,Z 439.989,A -85,B 0,C 180,E1 -11622.471,E2 -11622.471} C_VEL
LIN {X 0,Y 391.178,Z 430.82,A -85,B 0,C 180,E1 -11623.706,E2 -11623.706} C_VEL
LIN {X 0,Y 391.968,Z 419.551,A -85,B 0,C 180,E1 -11624.933,E2 -11624.933} C_VEL
LIN {X 0,Y 392.663,Z 409.147,A -85,B 0,C 180,E1 -11625.836,E2 -11625.836} C_VEL
LIN {X 0,Y 393.512,Z 396.708,A -85,B 0,C 180,E1 -11626.667,E2 -11626.667} C_VEL
LIN {X 0,Y 394.236,Z 383.594,A -85,B 0,C 180,E1 -11627.303,E2 -11627.303} C_VEL
LIN {X 0,Y 394.726,Z 370.705,A -85,B 0,C 180,E1 -11627.715,E2 -11627.715} C_VEL
LIN {X 0,Y 395.592,Z 293.501,A -85,B 0,C 180,E1 -11629.13,E2 -11629.13} C_VEL
LIN {X 0,Y 391.451,Z 262.744,A -85,B 0,C 180,E1 -11629.902,E2 -11629.902} C_VEL
LIN {X 0,Y 392.643,Z 244.878,A -85,B 0,C 180,E1 -11633.449,E2 -11633.449} C_VEL
LIN {X 0,Y 393.093,Z 236.547,A -85,B 0,C 180,E1 -11635.122,E2 -11635.122} C_VEL
LIN {X 0,Y 391.038,Z 225.247,A -85,B 0,C 180,E1 -11637.563,E2 -11637.563} C_VEL
LIN {X 0,Y 390.148,Z 220.889,A -85,B 0,C 180,E1 -11638.549,E2 -11638.549} C_VEL
LIN {X 0,Y 390.025,Z 220.899,A -85,B 0,C 180,E1 -11642.717,E2 -11642.717} C_VEL
LIN {X 0,Y 390.036,Z 220.902,A -85,B 0,C 180,E1 -11645.821,E2 -11645.821} C_VEL
LIN {X 0,Y 390.045,Z 220.896,A -85,B 0,C 180,E1 -11649.214,E2 -11649.214} C_VEL
LIN {X 0,Y 390.015,Z 220.901,A -85,B 0,C 180,E1 -11652.37,E2 -11652.37} C_VEL
LIN {X 0,Y 390.069,Z 220.896,A -85,B 0,C 180,E1 -11656.103,E2 -11656.103} C_VEL
LIN {X 0,Y 390.05,Z 220.896,A -85,B 0,C 180,E1 -11659.17,E2 -11659.17} C_VEL
LIN {X 0,Y 390.012,Z 220.9,A -85,B 0,C 180,E1 -11662.445,E2 -11662.445} C_VEL
LIN {X 0,Y 390.03,Z 220.9,A -85,B 0,C 180,E1 -11666.041,E2 -11666.041} C_VEL
LIN {X 0,Y 390.01,Z 220.903,A -85,B 0,C 180,E1 -11669.865,E2 -11669.865} C_VEL
LIN {X 0,Y 390.071,Z 220.896,A -85,B 0,C 180,E1 -11673.229,E2 -11673.229} C_VEL
LIN {X 0,Y 390.079,Z 220.892,A -85,B 0,C 180,E1 -11676.742,E2 -11676.742} C_VEL
LIN {X 0,Y 390.085,Z 220.892,A -85,B 0,C 180,E1 -11679.982,E2 -11679.982} C_VEL
LIN {X 0,Y 390.092,Z 220.896,A -85,B 0,C 180,E1 -11683.246,E2 -11683.246} C_VEL
LIN {X 0,Y 390.146,Z 220.883,A -85,B 0,C 180,E1 -11686.56,E2 -11686.56} C_VEL
LIN {X 0,Y 390.13,Z 220.888,A -85,B 0,C 180,E1 -11689.622,E2 -11689.622} C_VEL
LIN {X 0,Y 390.277,Z 220.869,A -85,B 0,C 180,E1 -11692.758,E2 -11692.758} C_VEL
LIN {X 0,Y 390.182,Z 220.882,A -85,B 0,C 180,E1 -11694.833,E2 -11694.833} C_VEL
LIN {X 0,Y 390.367,Z 220.855,A -85,B 0,C 180,E1 -11697.937,E2 -11697.937} C_VEL
LIN {X 0,Y 390.496,Z 220.839,A -85,B 0,C 180,E1 -11700,E2 -11700} C_VEL
LIN {X 0,Y 390.256,Z 220.875,A -85,B 0,C 180,E1 -11703.097,E2 -11703.097} C_VEL
LIN {X 0,Y 390.247,Z 220.87,A -85,B 0,C 180,E1 -11706.685,E2 -11706.685} C_VEL
LIN {X 0,Y 390.155,Z 220.884,A -85,B 0,C 180,E1 -11709.33,E2 -11709.33} C_VEL
LIN {X 0,Y 390.129,Z 220.888,A -85,B 0,C 180,E1 -11712.485,E2 -11712.485} C_VEL
LIN {X 0,Y 390.093,Z 220.889,A -85,B 0,C 180,E1 -11715.679,E2 -11715.679} C_VEL
LIN {X 0,Y 390.052,Z 220.899,A -85,B 0,C 180,E1 -11718.925,E2 -11718.925} C_VEL
LIN {X 0,Y 389.991,Z 220.905,A -85,B 0,C 180,E1 -11722.237,E2 -11722.237} C_VEL
LIN {X 0,Y 390.076,Z 220.892,A -85,B 0,C 180,E1 -11725.746,E2 -11725.746} C_VEL
LIN {X 0,Y 390.023,Z 220.899,A -85,B 0,C 180,E1 -11729.113,E2 -11729.113} C_VEL
LIN {X 0,Y 390.005,Z 220.904,A -85,B 0,C 180,E1 -11732.725,E2 -11732.725} C_VEL
LIN {X 0,Y 390.02,Z 220.9,A -85,B 0,C 180,E1 -11735.829,E2 -11735.829} C_VEL
LIN {X 0,Y 390.039,Z 220.896,A -85,B 0,C 180,E1 -11739.223,E2 -11739.223} C_VEL
LIN {X 0,Y 390.089,Z 220.896,A -85,B 0,C 180,E1 -11742.391,E2 -11742.391} C_VEL
LIN {X 0,Y 390.03,Z 220.897,A -85,B 0,C 180,E1 -11745.361,E2 -11745.361} C_VEL
LIN {X 0,Y 390.006,Z 220.907,A -85,B 0,C 180,E1 -11748.191,E2 -11748.191} C_VEL
LIN {X 0,Y 390.069,Z 220.893,A -85,B 0,C 180,E1 -11750.912,E2 -11750.912} C_VEL
LIN {X 0,Y 390.066,Z 220.893,A -85,B 0,C 180,E1 -11754.797,E2 -11754.797} C_VEL
LIN {X 0,Y 390.008,Z 220.902,A -85,B 0,C 180,E1 -11758.5,E2 -11758.5} C_VEL
LIN {X 0,Y 390.105,Z 220.893,A -85,B 0,C 180,E1 -11762.074,E2 -11762.074} C_VEL
LIN {X 0,Y 390.067,Z 220.895,A -85,B 0,C 180,E1 -11765.523,E2 -11765.523} C_VEL
LIN {X 0,Y 390.081,Z 220.895,A -85,B 0,C 180,E1 -11769.534,E2 -11769.534} C_VEL
LIN {X 0,Y 390.134,Z 220.886,A -85,B 0,C 180,E1 -11773.252,E2 -11773.252} C_VEL
LIN {X 0,Y 390.193,Z 220.877,A -85,B 0,C 180,E1 -11776.565,E2 -11776.565} C_VEL
LIN {X 0,Y 390.205,Z 220.955,A -85,B 0,C 180,E1 -11779.2,E2 -11779.2} C_VEL
LIN {X 0,Y 391.729,Z 229.225,A -85,B 0,C 180,E1 -11781.208,E2 -11781.208} C_VEL
LIN {X 0,Y 393.948,Z 239.601,A -85,B 0,C 180,E1 -11781.508,E2 -11781.508} C_VEL
LIN {X 0,Y 396.126,Z 252.417,A -85,B 0,C 180,E1 -11781.843,E2 -11781.843} C_VEL
LIN {X 0,Y 394.832,Z 336.965,A -85,B 0,C 180,E1 -11783.391,E2 -11783.391} C_VEL
LIN {X 0,Y 394.396,Z 350.727,A -85,B 0,C 180,E1 -11783.865,E2 -11783.865} C_VEL
LIN {X 0,Y 393.974,Z 361.942,A -85,B 0,C 180,E1 -11784.436,E2 -11784.436} C_VEL
LIN {X 0,Y 393.431,Z 374.06,A -85,B 0,C 180,E1 -11785.263,E2 -11785.263} C_VEL
LIN {X 0,Y 392.534,Z 385.589,A -85,B 0,C 180,E1 -11786.281,E2 -11786.281} C_VEL
LIN {X 0,Y 391.784,Z 395.935,A -85,B 0,C 180,E1 -11787.432,E2 -11787.432} C_VEL
LIN {X 0,Y 391.069,Z 405.263,A -85,B 0,C 180,E1 -11788.715,E2 -11788.715} C_VEL
LIN {X 0,Y 390.388,Z 414.259,A -85,B 0,C 180,E1 -11790.26,E2 -11790.26} C_VEL
LIN {X 0,Y 389.783,Z 421.53,A -85,B 0,C 180,E1 -11791.81,E2 -11791.81} C_VEL
LIN {X 0,Y 389.403,Z 428.179,A -85,B 0,C 180,E1 -11793.623,E2 -11793.623} C_VEL
LIN {X 0,Y 389.113,Z 432.586,A -85,B 0,C 180,E1 -11795.183,E2 -11795.183} C_VEL
LIN {X 0,Y 388.915,Z 436.206,A -85,B 0,C 180,E1 -11796.919,E2 -11796.919} C_VEL
LIN {X 0,Y 388.15,Z 437.595,A -85,B 0,C 180,E1 -11797.758,E2 -11797.758} C_VEL
LIN {X 0,Y 385.16,Z 439.298,A -85,B 0,C 180,E1 -11799.136,E2 -11799.136} C_VEL
LIN {X 0,Y 382.694,Z 440.149,A -85,B 0,C 180,E1 -11800.261,E2 -11800.261} C_VEL
LIN {X 0,Y 381.669,Z 440.476,A -85,B 0,C 180,E1 -11801.136,E2 -11801.136} C_VEL
LIN {X 0,Y 381.601,Z 440.495,A -85,B 0,C 180,E1 -11801.433,E2 -11801.433} C_VEL
LIN {X 0,Y 381.675,Z 440.29,A -85,B 0,C 180,E1 -11802.766,E2 -11802.766} C_VEL
LIN {X 0,Y 381.71,Z 439.652,A -85,B 0,C 180,E1 -11803.849,E2 -11803.849} C_VEL
LIN {X 0,Y 381.809,Z 438.613,A -85,B 0,C 180,E1 -11804.934,E2 -11804.934} C_VEL
LIN {X 0,Y 382.021,Z 437.104,A -85,B 0,C 180,E1 -11806.019,E2 -11806.019} C_VEL
LIN {X 0,Y 382.355,Z 434.013,A -85,B 0,C 180,E1 -11807.655,E2 -11807.655} C_VEL
LIN {X 0,Y 382.802,Z 429.802,A -85,B 0,C 180,E1 -11809.297,E2 -11809.297} C_VEL
LIN {X 0,Y 383.518,Z 423.879,A -85,B 0,C 180,E1 -11811.062,E2 -11811.062} C_VEL
LIN {X 0,Y 384.28,Z 417.428,A -85,B 0,C 180,E1 -11812.585,E2 -11812.585} C_VEL
LIN {X 0,Y 385.256,Z 409.628,A -85,B 0,C 180,E1 -11814.076,E2 -11814.076} C_VEL
LIN {X 0,Y 386.202,Z 400.674,A -85,B 0,C 180,E1 -11815.462,E2 -11815.462} C_VEL
LIN {X 0,Y 387.355,Z 389.642,A -85,B 0,C 180,E1 -11816.828,E2 -11816.828} C_VEL
LIN {X 0,Y 388.408,Z 379.22,A -85,B 0,C 180,E1 -11817.852,E2 -11817.852} C_VEL
LIN {X 0,Y 389.289,Z 366.89,A -85,B 0,C 180,E1 -11818.802,E2 -11818.802} C_VEL
LIN {X 0,Y 390.01,Z 355.127,A -85,B 0,C 180,E1 -11819.483,E2 -11819.483} C_VEL
LIN {X 0,Y 390.584,Z 342.736,A -85,B 0,C 180,E1 -11819.991,E2 -11819.991} C_VEL
LIN {X 0,Y 390.945,Z 329.534,A -85,B 0,C 180,E1 -11820.317,E2 -11820.317} C_VEL
LIN {X 0,Y 392.233,Z 252.574,A -85,B 0,C 180,E1 -11821.751,E2 -11821.751} C_VEL
LIN {X 0,Y 389.202,Z 240.659,A -85,B 0,C 180,E1 -11822.191,E2 -11822.191} C_VEL
LIN {X 0,Y 384.876,Z 229.945,A -85,B 0,C 180,E1 -11822.729,E2 -11822.729} C_VEL
LIN {X 0,Y 383.051,Z 221.773,A -85,B 0,C 180,E1 -11824.903,E2 -11824.903} C_VEL
LIN {X 0,Y 383.003,Z 221.783,A -85,B 0,C 180,E1 -11828.599,E2 -11828.599} C_VEL
LIN {X 0,Y 383.006,Z 221.779,A -85,B 0,C 180,E1 -11831.342,E2 -11831.342} C_VEL
LIN {X 0,Y 382.996,Z 221.771,A -85,B 0,C 180,E1 -11834.303,E2 -11834.303} C_VEL
LIN {X 0,Y 383.066,Z 221.768,A -85,B 0,C 180,E1 -11837.248,E2 -11837.248} C_VEL
LIN {X 0,Y 383.01,Z 221.776,A -85,B 0,C 180,E1 -11840.411,E2 -11840.411} C_VEL
LIN {X 0,Y 383.012,Z 221.778,A -85,B 0,C 180,E1 -11844.043,E2 -11844.043} C_VEL
LIN {X 0,Y 382.971,Z 221.782,A -85,B 0,C 180,E1 -11847.577,E2 -11847.577} C_VEL
LIN {X 0,Y 382.979,Z 221.779,A -85,B 0,C 180,E1 -11850.299,E2 -11850.299} C_VEL
LIN {X 0,Y 383.039,Z 221.764,A -85,B 0,C 180,E1 -11852.696,E2 -11852.696} C_VEL
LIN {X 0,Y 383.031,Z 221.771,A -85,B 0,C 180,E1 -11855.038,E2 -11855.038} C_VEL
LIN {X 0,Y 382.969,Z 221.778,A -85,B 0,C 180,E1 -11858.467,E2 -11858.467} C_VEL
LIN {X 0,Y 383.065,Z 221.77,A -85,B 0,C 180,E1 -11861.826,E2 -11861.826} C_VEL
LIN {X 0,Y 383.087,Z 221.759,A -85,B 0,C 180,E1 -11865.117,E2 -11865.117} C_VEL
LIN {X 0,Y 383.07,Z 221.762,A -85,B 0,C 180,E1 -11868.357,E2 -11868.357} C_VEL
LIN {X 0,Y 383.241,Z 221.744,A -85,B 0,C 180,E1 -11871.974,E2 -11871.974} C_VEL
LIN {X 0,Y 383.172,Z 221.75,A -85,B 0,C 180,E1 -11874.738,E2 -11874.738} C_VEL
LIN {X 0,Y 383.356,Z 221.723,A -85,B 0,C 180,E1 -11877.899,E2 -11877.899} C_VEL
LIN {X 0,Y 383.49,Z 221.713,A -85,B 0,C 180,E1 -11880,E2 -11880} C_VEL
LIN {X 0,Y 383.214,Z 221.744,A -85,B 0,C 180,E1 -11883.154,E2 -11883.154} C_VEL
LIN {X 0,Y 383.231,Z 221.745,A -85,B 0,C 180,E1 -11886.317,E2 -11886.317} C_VEL
LIN {X 0,Y 383.119,Z 221.761,A -85,B 0,C 180,E1 -11889.503,E2 -11889.503} C_VEL
LIN {X 0,Y 383.115,Z 221.756,A -85,B 0,C 180,E1 -11892.717,E2 -11892.717} C_VEL
LIN {X 0,Y 383.057,Z 221.765,A -85,B 0,C 180,E1 -11895.974,E2 -11895.974} C_VEL
LIN {X 0,Y 383.026,Z 221.772,A -85,B 0,C 180,E1 -11899.285,E2 -11899.285} C_VEL
LIN {X 0,Y 382.967,Z 221.779,A -85,B 0,C 180,E1 -11902.667,E2 -11902.667} C_VEL
LIN {X 0,Y 382.97,Z 221.773,A -85,B 0,C 180,E1 -11906.131,E2 -11906.131} C_VEL
LIN {X 0,Y 382.959,Z 221.774,A -85,B 0,C 180,E1 -11909.703,E2 -11909.703} C_VEL
LIN {X 0,Y 382.982,Z 221.771,A -85,B 0,C 180,E1 -11913.403,E2 -11913.403} C_VEL
LIN {X 0,Y 383.007,Z 221.776,A -85,B 0,C 180,E1 -11916.164,E2 -11916.164} C_VEL
LIN {X 0,Y 382.988,Z 221.769,A -85,B 0,C 180,E1 -11919.961,E2 -11919.961} C_VEL
LIN {X 0,Y 382.995,Z 221.775,A -85,B 0,C 180,E1 -11922.78,E2 -11922.78} C_VEL
LIN {X 0,Y 382.985,Z 221.776,A -85,B 0,C 180,E1 -11925.79,E2 -11925.79} C_VEL
LIN {X 0,Y 382.955,Z 221.776,A -85,B 0,C 180,E1 -11928.802,E2 -11928.802} C_VEL
LIN {X 0,Y 382.987,Z 221.774,A -85,B 0,C 180,E1 -11932.099,E2 -11932.099} C_VEL
LIN {X 0,Y 383.014,Z 221.774,A -85,B 0,C 180,E1 -11935.333,E2 -11935.333} C_VEL
LIN {X 0,Y 382.979,Z 221.782,A -85,B 0,C 180,E1 -11939.082,E2 -11939.082} C_VEL
LIN {X 0,Y 382.996,Z 221.875,A -85,B 0,C 180,E1 -11939.389,E2 -11939.389} C_VEL
LIN {X 0,Y 385.818,Z 233.802,A -85,B 0,C 180,E1 -11942.323,E2 -11942.323} C_VEL
LIN {X 0,Y 387.533,Z 243.084,A -85,B 0,C 180,E1 -11944.488,E2 -11944.488} C_VEL
LIN {X 0,Y 385.926,Z 259.974,A -85,B 0,C 180,E1 -11948.003,E2 -11948.003} C_VEL
LIN {X 0,Y 385.731,Z 261.909,A -85,B 0,C 180,E1 -11948.401,E2 -11948.401} C_VEL
LIN {X 0,Y 390.164,Z 285.524,A -85,B 0,C 180,E1 -11949.178,E2 -11949.178} C_VEL
LIN {X 0,Y 391.549,Z 295.222,A -85,B 0,C 180,E1 -11949.457,E2 -11949.457} C_VEL
LIN {X 0,Y 390.385,Z 370.718,A -85,B 0,C 180,E1 -11950.891,E2 -11950.891} C_VEL
LIN {X 0,Y 389.713,Z 383.853,A -85,B 0,C 180,E1 -11951.331,E2 -11951.331} C_VEL
LIN {X 0,Y 388.755,Z 396.578,A -85,B 0,C 180,E1 -11951.965,E2 -11951.965} C_VEL
LIN {X 0,Y 387.767,Z 407.905,A -85,B 0,C 180,E1 -11952.735,E2 -11952.735} C_VEL
LIN {X 0,Y 386.609,Z 419.583,A -85,B 0,C 180,E1 -11953.77,E2 -11953.77} C_VEL
LIN {X 0,Y 385.511,Z 430.09,A -85,B 0,C 180,E1 -11954.942,E2 -11954.942} C_VEL
LIN {X 0,Y 384.51,Z 439.587,A -85,B 0,C 180,E1 -11956.254,E2 -11956.254} C_VEL
LIN {X 0,Y 383.503,Z 448.754,A -85,B 0,C 180,E1 -11957.833,E2 -11957.833} C_VEL
LIN {X 0,Y 382.69,Z 456.156,A -85,B 0,C 180,E1 -11959.417,E2 -11959.417} C_VEL
LIN {X 0,Y 382.185,Z 462.12,A -85,B 0,C 180,E1 -11961.006,E2 -11961.006} C_VEL
LIN {X 0,Y 381.855,Z 466.849,A -85,B 0,C 180,E1 -11962.596,E2 -11962.596} C_VEL
LIN {X 0,Y 381.693,Z 469.843,A -85,B 0,C 180,E1 -11963.874,E2 -11963.874} C_VEL
LIN {X 0,Y 381.624,Z 473.109,A -85,B 0,C 180,E1 -11965.774,E2 -11965.774} C_VEL
LIN {X 0,Y 381.576,Z 474.356,A -85,B 0,C 180,E1 -11966.831,E2 -11966.831} C_VEL
LIN {X 0,Y 381.652,Z 475.183,A -85,B 0,C 180,E1 -11967.888,E2 -11967.888} C_VEL
LIN {X 0,Y 381.692,Z 475.592,A -85,B 0,C 180,E1 -11968.943,E2 -11968.943} C_VEL
LIN {X 0,Y 381.693,Z 475.245,A -85,B 0,C 180,E1 -11971.053,E2 -11971.053} C_VEL
LIN {X 0,Y 381.691,Z 474.466,A -85,B 0,C 180,E1 -11972.108,E2 -11972.108} C_VEL
LIN {X 0,Y 381.644,Z 471.616,A -85,B 0,C 180,E1 -11974.222,E2 -11974.222} C_VEL
LIN {X 0,Y 381.689,Z 467.591,A -85,B 0,C 180,E1 -11976.121,E2 -11976.121} C_VEL
LIN {X 0,Y 381.9,Z 462.249,A -85,B 0,C 180,E1 -11977.931,E2 -11977.931} C_VEL
LIN {X 0,Y 382.274,Z 455.08,A -85,B 0,C 180,E1 -11979.788,E2 -11979.788} C_VEL
LIN {X 0,Y 382.834,Z 447.279,A -85,B 0,C 180,E1 -11981.379,E2 -11981.379} C_VEL
LIN {X 0,Y 383.437,Z 439.282,A -85,B 0,C 180,E1 -11982.703,E2 -11982.703} C_VEL
LIN {X 0,Y 384.172,Z 429.518,A -85,B 0,C 180,E1 -11984.024,E2 -11984.024} C_VEL
LIN {X 0,Y 385.035,Z 418.665,A -85,B 0,C 180,E1 -11985.208,E2 -11985.208} C_VEL
LIN {X 0,Y 385.829,Z 408.117,A -85,B 0,C 180,E1 -11986.124,E2 -11986.124} C_VEL
LIN {X 0,Y 386.698,Z 395.407,A -85,B 0,C 180,E1 -11986.97,E2 -11986.97} C_VEL
LIN {X 0,Y 387.394,Z 382.718,A -85,B 0,C 180,E1 -11987.584,E2 -11987.584} C_VEL
LIN {X 0,Y 387.891,Z 369.299,A -85,B 0,C 180,E1 -11988.004,E2 -11988.004} C_VEL
LIN {X 0,Y 388.77,Z 294.259,A -85,B 0,C 180,E1 -11989.4,E2 -11989.4} C_VEL
LIN {X 0,Y 384.501,Z 262.474,A -85,B 0,C 180,E1 -11990.204,E2 -11990.204} C_VEL
LIN {X 0,Y 385.67,Z 245.521,A -85,B 0,C 180,E1 -11993.63,E2 -11993.63} C_VEL
LIN {X 0,Y 386.076,Z 237.265,A -85,B 0,C 180,E1 -11995.322,E2 -11995.322} C_VEL
LIN {X 0,Y 383.614,Z 224.241,A -85,B 0,C 180,E1 -11998.204,E2 -11998.204} C_VEL
LIN {X 0,Y 383.078,Z 221.769,A -85,B 0,C 180,E1 -11998.784,E2 -11998.784} C_VEL
LIN {X 0,Y 382.969,Z 221.78,A -85,B 0,C 180,E1 -12002.418,E2 -12002.418} C_VEL
LIN {X 0,Y 383.004,Z 221.779,A -85,B 0,C 180,E1 -12005.951,E2 -12005.951} C_VEL
LIN {X 0,Y 382.991,Z 221.777,A -85,B 0,C 180,E1 -12009.582,E2 -12009.582} C_VEL
LIN {X 0,Y 382.98,Z 221.776,A -85,B 0,C 180,E1 -12012.774,E2 -12012.774} C_VEL
LIN {X 0,Y 383.005,Z 221.779,A -85,B 0,C 180,E1 -12015.79,E2 -12015.79} C_VEL
LIN {X 0,Y 383.013,Z 221.771,A -85,B 0,C 180,E1 -12018.782,E2 -12018.782} C_VEL
LIN {X 0,Y 382.969,Z 221.78,A -85,B 0,C 180,E1 -12022.092,E2 -12022.092} C_VEL
LIN {X 0,Y 382.981,Z 221.779,A -85,B 0,C 180,E1 -12025.328,E2 -12025.328} C_VEL
LIN {X 0,Y 382.945,Z 221.782,A -85,B 0,C 180,E1 -12029.078,E2 -12029.078} C_VEL
LIN {X 0,Y 383.015,Z 221.771,A -85,B 0,C 180,E1 -12032.695,E2 -12032.695} C_VEL
LIN {X 0,Y 383.004,Z 221.773,A -85,B 0,C 180,E1 -12036.191,E2 -12036.191} C_VEL
LIN {X 0,Y 383.038,Z 221.773,A -85,B 0,C 180,E1 -12039.597,E2 -12039.597} C_VEL
LIN {X 0,Y 383.058,Z 221.768,A -85,B 0,C 180,E1 -12042.929,E2 -12042.929} C_VEL
LIN {X 0,Y 383.078,Z 221.764,A -85,B 0,C 180,E1 -12046.462,E2 -12046.462} C_VEL
LIN {X 0,Y 383.092,Z 221.766,A -85,B 0,C 180,E1 -12049.429,E2 -12049.429} C_VEL
LIN {X 0,Y 383.23,Z 221.746,A -85,B 0,C 180,E1 -12052.625,E2 -12052.625} C_VEL
LIN {X 0,Y 383.155,Z 221.756,A -85,B 0,C 180,E1 -12054.738,E2 -12054.738} C_VEL
LIN {X 0,Y 383.335,Z 221.732,A -85,B 0,C 180,E1 -12057.899,E2 -12057.899} C_VEL
LIN {X 0,Y 383.466,Z 221.715,A -85,B 0,C 180,E1 -12060,E2 -12060} C_VEL
LIN {X 0,Y 383.193,Z 221.754,A -85,B 0,C 180,E1 -12063.154,E2 -12063.154} C_VEL
LIN {X 0,Y 383.206,Z 221.747,A -85,B 0,C 180,E1 -12066.678,E2 -12066.678} C_VEL
LIN {X 0,Y 383.103,Z 221.761,A -85,B 0,C 180,E1 -12069.503,E2 -12069.503} C_VEL
LIN {X 0,Y 383.092,Z 221.767,A -85,B 0,C 180,E1 -12072.718,E2 -12072.718} C_VEL
LIN {X 0,Y 383.035,Z 221.769,A -85,B 0,C 180,E1 -12075.976,E2 -12075.976} C_VEL
LIN {X 0,Y 383.004,Z 221.774,A -85,B 0,C 180,E1 -12079.287,E2 -12079.287} C_VEL
LIN {X 0,Y 382.946,Z 221.786,A -85,B 0,C 180,E1 -12082.669,E2 -12082.669} C_VEL
LIN {X 0,Y 383.038,Z 221.77,A -85,B 0,C 180,E1 -12086.127,E2 -12086.127} C_VEL
LIN {X 0,Y 383.002,Z 221.779,A -85,B 0,C 180,E1 -12088.496,E2 -12088.496} C_VEL
LIN {X 0,Y 382.971,Z 221.78,A -85,B 0,C 180,E1 -12092.154,E2 -12092.154} C_VEL
LIN {X 0,Y 382.982,Z 221.779,A -85,B 0,C 180,E1 -12094.672,E2 -12094.672} C_VEL
LIN {X 0,Y 382.967,Z 221.779,A -85,B 0,C 180,E1 -12097.908,E2 -12097.908} C_VEL
LIN {X 0,Y 383.015,Z 221.771,A -85,B 0,C 180,E1 -12101.344,E2 -12101.344} C_VEL
LIN {X 0,Y 383.002,Z 221.779,A -85,B 0,C 180,E1 -12104.313,E2 -12104.313} C_VEL
LIN {X 0,Y 382.986,Z 221.775,A -85,B 0,C 180,E1 -12107.245,E2 -12107.245} C_VEL
LIN {X 0,Y 382.993,Z 221.778,A -85,B 0,C 180,E1 -12110.418,E2 -12110.418} C_VEL
LIN {X 0,Y 383.006,Z 221.779,A -85,B 0,C 180,E1 -12114.049,E2 -12114.049} C_VEL
LIN {X 0,Y 382.971,Z 221.779,A -85,B 0,C 180,E1 -12117.583,E2 -12117.583} C_VEL
LIN {X 0,Y 382.978,Z 221.779,A -85,B 0,C 180,E1 -12120.304,E2 -12120.304} C_VEL
LIN {X 0,Y 383.069,Z 221.77,A -85,B 0,C 180,E1 -12124.025,E2 -12124.025} C_VEL
LIN {X 0,Y 382.983,Z 221.777,A -85,B 0,C 180,E1 -12127.338,E2 -12127.338} C_VEL
LIN {X 0,Y 383.052,Z 221.767,A -85,B 0,C 180,E1 -12130.72,E2 -12130.72} C_VEL
LIN {X 0,Y 383.077,Z 221.767,A -85,B 0,C 180,E1 -12134.03,E2 -12134.03} C_VEL
LIN {X 0,Y 383.135,Z 221.759,A -85,B 0,C 180,E1 -12137.287,E2 -12137.287} C_VEL
LIN {X 0,Y 383.148,Z 221.893,A -85,B 0,C 180,E1 -12138.999,E2 -12138.999} C_VEL
LIN {X 0,Y 384.603,Z 229.553,A -85,B 0,C 180,E1 -12140.89,E2 -12140.89} C_VEL
LIN {X 0,Y 386.496,Z 236.922,A -85,B 0,C 180,E1 -12141.122,E2 -12141.122} C_VEL
LIN {X 0,Y 389.331,Z 252.535,A -85,B 0,C 180,E1 -12141.549,E2 -12141.549} C_VEL
LIN {X 0,Y 388,Z 336.72,A -85,B 0,C 180,E1 -12143.11,E2 -12143.11} C_VEL
LIN {X 0,Y 387.56,Z 349.926,A -85,B 0,C 180,E1 -12143.56,E2 -12143.56} C_VEL
LIN {X 0,Y 387.136,Z 361.424,A -85,B 0,C 180,E1 -12144.142,E2 -12144.142} C_VEL
LIN {X 0,Y 386.655,Z 372.91,A -85,B 0,C 180,E1 -12144.919,E2 -12144.919} C_VEL
LIN {X 0,Y 385.832,Z 383.484,A -85,B 0,C 180,E1 -12145.824,E2 -12145.824} C_VEL
LIN {X 0,Y 384.992,Z 394.266,A -85,B 0,C 180,E1 -12146.994,E2 -12146.994} C_VEL
LIN {X 0,Y 384.265,Z 403.07,A -85,B 0,C 180,E1 -12148.168,E2 -12148.168} C_VEL
LIN {X 0,Y 383.542,Z 412.627,A -85,B 0,C 180,E1 -12149.74,E2 -12149.74} C_VEL
LIN {X 0,Y 382.835,Z 420.263,A -85,B 0,C 180,E1 -12151.317,E2 -12151.317} C_VEL
LIN {X 0,Y 382.41,Z 427.28,A -85,B 0,C 180,E1 -12153.162,E2 -12153.162} C_VEL
LIN {X 0,Y 382.06,Z 431.967,A -85,B 0,C 180,E1 -12154.75,E2 -12154.75} C_VEL
LIN {X 0,Y 381.908,Z 435.702,A -85,B 0,C 180,E1 -12156.418,E2 -12156.418} C_VEL
LIN {X 0,Y 381.787,Z 437.392,A -85,B 0,C 180,E1 -12157.405,E2 -12157.405} C_VEL
LIN {X 0,Y 381.666,Z 438.776,A -85,B 0,C 180,E1 -12158.472,E2 -12158.472} C_VEL
LIN {X 0,Y 381.593,Z 440.36,A -85,B 0,C 180,E1 -12160.614,E2 -12160.614} C_VEL
LIN {X 0,Y 381.601,Z 440.495,A -85,B 0,C 180,E1 -12161.433,E2 -12161.433} C_VEL
LIN {X 0,Y 380.974,Z 440.507,A -85,B 0,C 180,E1 -12162.314,E2 -12162.314} C_VEL
LIN {X 0,Y 378.162,Z 439.95,A -85,B 0,C 180,E1 -12163.747,E2 -12163.747} C_VEL
LIN {X 0,Y 375.841,Z 439.04,A -85,B 0,C 180,E1 -12164.898,E2 -12164.898} C_VEL
LIN {X 0,Y 374.953,Z 438.008,A -85,B 0,C 180,E1 -12165.78,E2 -12165.78} C_VEL
LIN {X 0,Y 374.94,Z 437.536,A -85,B 0,C 180,E1 -12166.076,E2 -12166.076} C_VEL
LIN {X 0,Y 375.364,Z 433.987,A -85,B 0,C 180,E1 -12167.995,E2 -12167.995} C_VEL
LIN {X 0,Y 375.872,Z 429.667,A -85,B 0,C 180,E1 -12169.668,E2 -12169.668} C_VEL
LIN {X 0,Y 376.615,Z 423.96,A -85,B 0,C 180,E1 -12171.374,E2 -12171.374} C_VEL
LIN {X 0,Y 377.476,Z 417.046,A -85,B 0,C 180,E1 -12173.016,E2 -12173.016} C_VEL
LIN {X 0,Y 378.524,Z 409.082,A -85,B 0,C 180,E1 -12174.525,E2 -12174.525} C_VEL
LIN {X 0,Y 379.552,Z 399.886,A -85,B 0,C 180,E1 -12175.941,E2 -12175.941} C_VEL
LIN {X 0,Y 380.667,Z 389.848,A -85,B 0,C 180,E1 -12177.189,E2 -12177.189} C_VEL
LIN {X 0,Y 381.834,Z 378.511,A -85,B 0,C 180,E1 -12178.307,E2 -12178.307} C_VEL
LIN {X 0,Y 382.745,Z 365.984,A -85,B 0,C 180,E1 -12179.267,E2 -12179.267} C_VEL
LIN {X 0,Y 383.51,Z 354.143,A -85,B 0,C 180,E1 -12179.941,E2 -12179.941} C_VEL
LIN {X 0,Y 384.066,Z 341.828,A -85,B 0,C 180,E1 -12180.43,E2 -12180.43} C_VEL
LIN {X 0,Y 384.462,Z 326.489,A -85,B 0,C 180,E1 -12180.786,E2 -12180.786} C_VEL
LIN {X 0,Y 385.748,Z 253.628,A -85,B 0,C 180,E1 -12182.165,E2 -12182.165} C_VEL
LIN {X 0,Y 383.053,Z 243.22,A -85,B 0,C 180,E1 -12182.563,E2 -12182.563} C_VEL
LIN {X 0,Y 377.736,Z 230.301,A -85,B 0,C 180,E1 -12183.234,E2 -12183.234} C_VEL
LIN {X 0,Y 376.013,Z 222.649,A -85,B 0,C 180,E1 -12185.354,E2 -12185.354} C_VEL
LIN {X 0,Y 375.963,Z 222.656,A -85,B 0,C 180,E1 -12189.461,E2 -12189.461} C_VEL
LIN {X 0,Y 375.955,Z 222.661,A -85,B 0,C 180,E1 -12192.295,E2 -12192.295} C_VEL
LIN {X 0,Y 375.967,Z 222.652,A -85,B 0,C 180,E1 -12195.26,E2 -12195.26} C_VEL
LIN {X 0,Y 375.979,Z 222.654,A -85,B 0,C 180,E1 -12198.388,E2 -12198.388} C_VEL
LIN {X 0,Y 375.954,Z 222.655,A -85,B 0,C 180,E1 -12201.91,E2 -12201.91} C_VEL
LIN {X 0,Y 375.966,Z 222.651,A -85,B 0,C 180,E1 -12205.331,E2 -12205.331} C_VEL
LIN {X 0,Y 375.943,Z 222.651,A -85,B 0,C 180,E1 -12208.436,E2 -12208.436} C_VEL
LIN {X 0,Y 375.979,Z 222.646,A -85,B 0,C 180,E1 -12212.14,E2 -12212.14} C_VEL
LIN {X 0,Y 375.986,Z 222.648,A -85,B 0,C 180,E1 -12214.537,E2 -12214.537} C_VEL
LIN {X 0,Y 375.935,Z 222.657,A -85,B 0,C 180,E1 -12218.044,E2 -12218.044} C_VEL
LIN {X 0,Y 375.998,Z 222.645,A -85,B 0,C 180,E1 -12221.472,E2 -12221.472} C_VEL
LIN {X 0,Y 376.036,Z 222.636,A -85,B 0,C 180,E1 -12224.831,E2 -12224.831} C_VEL
LIN {X 0,Y 376.023,Z 222.64,A -85,B 0,C 180,E1 -12228.136,E2 -12228.136} C_VEL
LIN {X 0,Y 376.197,Z 222.622,A -85,B 0,C 180,E1 -12231.918,E2 -12231.918} C_VEL
LIN {X 0,Y 376.145,Z 222.625,A -85,B 0,C 180,E1 -12234.639,E2 -12234.639} C_VEL
LIN {X 0,Y 376.322,Z 222.599,A -85,B 0,C 180,E1 -12237.859,E2 -12237.859} C_VEL
LIN {X 0,Y 376.46,Z 222.589,A -85,B 0,C 180,E1 -12240,E2 -12240} C_VEL
LIN {X 0,Y 376.152,Z 222.624,A -85,B 0,C 180,E1 -12243.213,E2 -12243.213} C_VEL
LIN {X 0,Y 376.19,Z 222.622,A -85,B 0,C 180,E1 -12246.436,E2 -12246.436} C_VEL
LIN {X 0,Y 376.09,Z 222.635,A -85,B 0,C 180,E1 -12249.682,E2 -12249.682} C_VEL
LIN {X 0,Y 376.067,Z 222.637,A -85,B 0,C 180,E1 -12253.658,E2 -12253.658} C_VEL
LIN {X 0,Y 376.011,Z 222.642,A -85,B 0,C 180,E1 -12257.401,E2 -12257.401} C_VEL
LIN {X 0,Y 375.959,Z 222.649,A -85,B 0,C 180,E1 -12260.833,E2 -12260.833} C_VEL
LIN {X 0,Y 375.941,Z 222.656,A -85,B 0,C 180,E1 -12264.285,E2 -12264.285} C_VEL
LIN {X 0,Y 375.914,Z 222.658,A -85,B 0,C 180,E1 -12267.865,E2 -12267.865} C_VEL
LIN {X 0,Y 375.92,Z 222.657,A -85,B 0,C 180,E1 -12270.69,E2 -12270.69} C_VEL
LIN {X 0,Y 375.941,Z 222.65,A -85,B 0,C 180,E1 -12274.113,E2 -12274.113} C_VEL
LIN {X 0,Y 375.934,Z 222.649,A -85,B 0,C 180,E1 -12276.743,E2 -12276.743} C_VEL
LIN {X 0,Y 375.968,Z 222.643,A -85,B 0,C 180,E1 -12279.97,E2 -12279.97} C_VEL
LIN {X 0,Y 375.918,Z 222.658,A -85,B 0,C 180,E1 -12283.768,E2 -12283.768} C_VEL
LIN {X 0,Y 375.925,Z 222.656,A -85,B 0,C 180,E1 -12286.812,E2 -12286.812} C_VEL
LIN {X 0,Y 375.927,Z 222.657,A -85,B 0,C 180,E1 -12290.535,E2 -12290.535} C_VEL
LIN {X 0,Y 375.957,Z 222.656,A -85,B 0,C 180,E1 -12293.497,E2 -12293.497} C_VEL
LIN {X 0,Y 375.957,Z 222.658,A -85,B 0,C 180,E1 -12295.89,E2 -12295.89} C_VEL
LIN {X 0,Y 375.971,Z 222.791,A -85,B 0,C 180,E1 -12298.966,E2 -12298.966} C_VEL
LIN {X 0,Y 378.891,Z 235.124,A -85,B 0,C 180,E1 -12302.073,E2 -12302.073} C_VEL
LIN {X 0,Y 380.649,Z 244.404,A -85,B 0,C 180,E1 -12304.287,E2 -12304.287} C_VEL
LIN {X 0,Y 379.116,Z 260.011,A -85,B 0,C 180,E1 -12307.6,E2 -12307.6} C_VEL
LIN {X 0,Y 378.987,Z 261.582,A -85,B 0,C 180,E1 -12307.932,E2 -12307.932} C_VEL
LIN {X 0,Y 383.744,Z 286.964,A -85,B 0,C 180,E1 -12308.784,E2 -12308.784} C_VEL
LIN {X 0,Y 385.069,Z 296.39,A -85,B 0,C 180,E1 -12309.062,E2 -12309.062} C_VEL
LIN {X 0,Y 383.796,Z 371.174,A -85,B 0,C 180,E1 -12310.511,E2 -12310.511} C_VEL
LIN {X 0,Y 383.089,Z 384.132,A -85,B 0,C 180,E1 -12310.961,E2 -12310.961} C_VEL
LIN {X 0,Y 382.054,Z 397.235,A -85,B 0,C 180,E1 -12311.638,E2 -12311.638} C_VEL
LIN {X 0,Y 381.013,Z 408.285,A -85,B 0,C 180,E1 -12312.419,E2 -12312.419} C_VEL
LIN {X 0,Y 379.814,Z 419.816,A -85,B 0,C 180,E1 -12313.471,E2 -12313.471} C_VEL
LIN {X 0,Y 378.664,Z 430.219,A -85,B 0,C 180,E1 -12314.663,E2 -12314.663} C_VEL
LIN {X 0,Y 377.604,Z 439.619,A -85,B 0,C 180,E1 -12315.997,E2 -12315.997} C_VEL
LIN {X 0,Y 376.551,Z 448.712,A -85,B 0,C 180,E1 -12317.605,E2 -12317.605} C_VEL
LIN {X 0,Y 375.667,Z 456.063,A -85,B 0,C 180,E1 -12319.217,E2 -12319.217} C_VEL
LIN {X 0,Y 375.143,Z 461.982,A -85,B 0,C 180,E1 -12320.836,E2 -12320.836} C_VEL
LIN {X 0,Y 374.77,Z 466.67,A -85,B 0,C 180,E1 -12322.456,E2 -12322.456} C_VEL
LIN {X 0,Y 374.587,Z 469.965,A -85,B 0,C 180,E1 -12323.927,E2 -12323.927} C_VEL
LIN {X 0,Y 374.55,Z 472.857,A -85,B 0,C 180,E1 -12325.694,E2 -12325.694} C_VEL
LIN {X 0,Y 374.488,Z 474.085,A -85,B 0,C 180,E1 -12326.771,E2 -12326.771} C_VEL
LIN {X 0,Y 374.551,Z 474.88,A -85,B 0,C 180,E1 -12327.848,E2 -12327.848} C_VEL
LIN {X 0,Y 374.624,Z 475.273,A -85,B 0,C 180,E1 -12328.923,E2 -12328.923} C_VEL
LIN {X 0,Y 374.626,Z 474.893,A -85,B 0,C 180,E1 -12331.073,E2 -12331.073} C_VEL
LIN {X 0,Y 374.592,Z 474.079,A -85,B 0,C 180,E1 -12332.148,E2 -12332.148} C_VEL
LIN {X 0,Y 374.575,Z 471.195,A -85,B 0,C 180,E1 -12334.302,E2 -12334.302} C_VEL
LIN {X 0,Y 374.591,Z 467.503,A -85,B 0,C 180,E1 -12336.078,E2 -12336.078} C_VEL
LIN {X 0,Y 374.761,Z 463.461,A -85,B 0,C 180,E1 -12337.54,E2 -12337.54} C_VEL
LIN {X 0,Y 375.014,Z 457.833,A -85,B 0,C 180,E1 -12339.163,E2 -12339.163} C_VEL
LIN {X 0,Y 375.454,Z 450.795,A -85,B 0,C 180,E1 -12340.786,E2 -12340.786} C_VEL
LIN {X 0,Y 376.249,Z 441.974,A -85,B 0,C 180,E1 -12342.401,E2 -12342.401} C_VEL
LIN {X 0,Y 377.059,Z 431.933,A -85,B 0,C 180,E1 -12343.882,E2 -12343.882} C_VEL
LIN {X 0,Y 377.84,Z 421.695,A -85,B 0,C 180,E1 -12345.091,E2 -12345.091} C_VEL
LIN {X 0,Y 378.676,Z 410.315,A -85,B 0,C 180,E1 -12346.16,E2 -12346.16} C_VEL
LIN {X 0,Y 379.557,Z 398.529,A -85,B 0,C 180,E1 -12347.021,E2 -12347.021} C_VEL
LIN {X 0,Y 380.322,Z 385.661,A -85,B 0,C 180,E1 -12347.714,E2 -12347.714} C_VEL
LIN {X 0,Y 380.965,Z 371.927,A -85,B 0,C 180,E1 -12348.204,E2 -12348.204} C_VEL
LIN {X 0,Y 381.764,Z 318.062,A -85,B 0,C 180,E1 -12349.243,E2 -12349.243} C_VEL
LIN {X 0,Y 381.883,Z 294.116,A -85,B 0,C 180,E1 -12349.7,E2 -12349.7} C_VEL
LIN {X 0,Y 377.574,Z 262.073,A -85,B 0,C 180,E1 -12350.541,E2 -12350.541} C_VEL
LIN {X 0,Y 378.797,Z 244.875,A -85,B 0,C 180,E1 -12354.086,E2 -12354.086} C_VEL
LIN {X 0,Y 379.171,Z 239.378,A -85,B 0,C 180,E1 -12355.229,E2 -12355.229} C_VEL
LIN {X 0,Y 377.659,Z 230.53,A -85,B 0,C 180,E1 -12357.2,E2 -12357.2} C_VEL
LIN {X 0,Y 376.023,Z 222.647,A -85,B 0,C 180,E1 -12359.034,E2 -12359.034} C_VEL
LIN {X 0,Y 375.932,Z 222.654,A -85,B 0,C 180,E1 -12362.824,E2 -12362.824} C_VEL
LIN {X 0,Y 375.938,Z 222.654,A -85,B 0,C 180,E1 -12365.411,E2 -12365.411} C_VEL
LIN {X 0,Y 375.951,Z 222.654,A -85,B 0,C 180,E1 -12368.266,E2 -12368.266} C_VEL
LIN {X 0,Y 375.908,Z 222.66,A -85,B 0,C 180,E1 -12371.596,E2 -12371.596} C_VEL
LIN {X 0,Y 375.947,Z 222.653,A -85,B 0,C 180,E1 -12375.257,E2 -12375.257} C_VEL
LIN {X 0,Y 375.959,Z 222.651,A -85,B 0,C 180,E1 -12378.386,E2 -12378.386} C_VEL
LIN {X 0,Y 375.934,Z 222.658,A -85,B 0,C 180,E1 -12381.908,E2 -12381.908} C_VEL
LIN {X 0,Y 375.943,Z 222.655,A -85,B 0,C 180,E1 -12385.329,E2 -12385.329} C_VEL
LIN {X 0,Y 375.92,Z 222.655,A -85,B 0,C 180,E1 -12388.434,E2 -12388.434} C_VEL
LIN {X 0,Y 375.955,Z 222.652,A -85,B 0,C 180,E1 -12392.138,E2 -12392.138} C_VEL
LIN {X 0,Y 375.964,Z 222.65,A -85,B 0,C 180,E1 -12394.536,E2 -12394.536} C_VEL
LIN {X 0,Y 375.98,Z 222.649,A -85,B 0,C 180,E1 -12398.047,E2 -12398.047} C_VEL
LIN {X 0,Y 375.986,Z 222.652,A -85,B 0,C 180,E1 -12401.472,E2 -12401.472} C_VEL
LIN {X 0,Y 376.013,Z 222.645,A -85,B 0,C 180,E1 -12404.831,E2 -12404.831} C_VEL
LIN {X 0,Y 376.009,Z 222.644,A -85,B 0,C 180,E1 -12408.135,E2 -12408.135} C_VEL
LIN {X 0,Y 376.211,Z 222.619,A -85,B 0,C 180,E1 -12411.874,E2 -12411.874} C_VEL
LIN {X 0,Y 376.128,Z 222.631,A -85,B 0,C 180,E1 -12414.639,E2 -12414.639} C_VEL
LIN {X 0,Y 376.302,Z 222.608,A -85,B 0,C 180,E1 -12417.859,E2 -12417.859} C_VEL
LIN {X 0,Y 376.436,Z 222.591,A -85,B 0,C 180,E1 -12420,E2 -12420} C_VEL
LIN {X 0,Y 376.131,Z 222.633,A -85,B 0,C 180,E1 -12423.214,E2 -12423.214} C_VEL
LIN {X 0,Y 376.17,Z 222.624,A -85,B 0,C 180,E1 -12426.668,E2 -12426.668} C_VEL
LIN {X 0,Y 376.071,Z 222.636,A -85,B 0,C 180,E1 -12429.683,E2 -12429.683} C_VEL
LIN {X 0,Y 376.042,Z 222.64,A -85,B 0,C 180,E1 -12433.659,E2 -12433.659} C_VEL
LIN {X 0,Y 375.997,Z 222.646,A -85,B 0,C 180,E1 -12437.609,E2 -12437.609} C_VEL
LIN {X 0,Y 375.935,Z 222.658,A -85,B 0,C 180,E1 -12440.835,E2 -12440.835} C_VEL
LIN {X 0,Y 375.945,Z 222.655,A -85,B 0,C 180,E1 -12444.285,E2 -12444.285} C_VEL
LIN {X 0,Y 375.978,Z 222.654,A -85,B 0,C 180,E1 -12446.656,E2 -12446.656} C_VEL
LIN {X 0,Y 375.933,Z 222.655,A -85,B 0,C 180,E1 -12449.083,E2 -12449.083} C_VEL
LIN {X 0,Y 375.912,Z 222.659,A -85,B 0,C 180,E1 -12452.832,E2 -12452.832} C_VEL
LIN {X 0,Y 375.921,Z 222.655,A -85,B 0,C 180,E1 -12455.42,E2 -12455.42} C_VEL
LIN {X 0,Y 375.942,Z 222.658,A -85,B 0,C 180,E1 -12458.275,E2 -12458.275} C_VEL
LIN {X 0,Y 375.959,Z 222.651,A -85,B 0,C 180,E1 -12461.614,E2 -12461.614} C_VEL
LIN {X 0,Y 375.939,Z 222.653,A -85,B 0,C 180,E1 -12465.267,E2 -12465.267} C_VEL
LIN {X 0,Y 375.916,Z 222.656,A -85,B 0,C 180,E1 -12469.137,E2 -12469.137} C_VEL
LIN {X 0,Y 375.943,Z 222.656,A -85,B 0,C 180,E1 -12471.916,E2 -12471.916} C_VEL
LIN {X 0,Y 375.962,Z 222.65,A -85,B 0,C 180,E1 -12475.337,E2 -12475.337} C_VEL
LIN {X 0,Y 375.942,Z 222.655,A -85,B 0,C 180,E1 -12478.442,E2 -12478.442} C_VEL
LIN {X 0,Y 375.971,Z 222.653,A -85,B 0,C 180,E1 -12482.145,E2 -12482.145} C_VEL
LIN {X 0,Y 375.995,Z 222.647,A -85,B 0,C 180,E1 -12484.543,E2 -12484.543} C_VEL
LIN {X 0,Y 375.949,Z 222.656,A -85,B 0,C 180,E1 -12488.049,E2 -12488.049} C_VEL
LIN {X 0,Y 375.997,Z 222.649,A -85,B 0,C 180,E1 -12491.477,E2 -12491.477} C_VEL
LIN {X 0,Y 376.055,Z 222.638,A -85,B 0,C 180,E1 -12494.836,E2 -12494.836} C_VEL
LIN {X 0,Y 376.048,Z 222.645,A -85,B 0,C 180,E1 -12498.14,E2 -12498.14} C_VEL
LIN {X 0,Y 376.083,Z 222.693,A -85,B 0,C 180,E1 -12498.756,E2 -12498.756} C_VEL
LIN {X 0,Y 377.471,Z 229.815,A -85,B 0,C 180,E1 -12500.545,E2 -12500.545} C_VEL
LIN {X 0,Y 379.728,Z 237.918,A -85,B 0,C 180,E1 -12500.828,E2 -12500.828} C_VEL
LIN {X 0,Y 382.529,Z 253.633,A -85,B 0,C 180,E1 -12501.263,E2 -12501.263} C_VEL
LIN {X 0,Y 381.138,Z 337.604,A -85,B 0,C 180,E1 -12502.853,E2 -12502.853} C_VEL
LIN {X 0,Y 380.691,Z 351.361,A -85,B 0,C 180,E1 -12503.344,E2 -12503.344} C_VEL
LIN {X 0,Y 380.169,Z 363.155,A -85,B 0,C 180,E1 -12503.967,E2 -12503.967} C_VEL
LIN {X 0,Y 379.602,Z 375.096,A -85,B 0,C 180,E1 -12504.824,E2 -12504.824} C_VEL
LIN {X 0,Y 378.645,Z 386.557,A -85,B 0,C 180,E1 -12505.878,E2 -12505.878} C_VEL
LIN {X 0,Y 377.842,Z 396.848,A -85,B 0,C 180,E1 -12507.07,E2 -12507.07} C_VEL
LIN {X 0,Y 377.055,Z 406.117,A -85,B 0,C 180,E1 -12508.4,E2 -12508.4} C_VEL
LIN {X 0,Y 376.348,Z 415.075,A -85,B 0,C 180,E1 -12510.002,E2 -12510.002} C_VEL
LIN {X 0,Y 375.692,Z 422.32,A -85,B 0,C 180,E1 -12511.61,E2 -12511.61} C_VEL
LIN {X 0,Y 375.318,Z 428.112,A -85,B 0,C 180,E1 -12513.222,E2 -12513.222} C_VEL
LIN {X 0,Y 374.975,Z 432.689,A -85,B 0,C 180,E1 -12514.84,E2 -12514.84} C_VEL
LIN {X 0,Y 374.826,Z 436.17,A -85,B 0,C 180,E1 -12516.461,E2 -12516.461} C_VEL
LIN {X 0,Y 374.669,Z 437.927,A -85,B 0,C 180,E1 -12517.546,E2 -12517.546} C_VEL
LIN {X 0,Y 374.577,Z 439.263,A -85,B 0,C 180,E1 -12518.634,E2 -12518.634} C_VEL
LIN {X 0,Y 374.476,Z 440.208,A -85,B 0,C 180,E1 -12519.725,E2 -12519.725} C_VEL
LIN {X 0,Y 374.515,Z 440.802,A -85,B 0,C 180,E1 -12521.442,E2 -12521.442} C_VEL
LIN {X 0,Y 374.595,Z 440.553,A -85,B 0,C 180,E1 -12523.012,E2 -12523.012} C_VEL
LIN {X 0,Y 374.649,Z 439.868,A -85,B 0,C 180,E1 -12524.115,E2 -12524.115} C_VEL
LIN {X 0,Y 374.94,Z 437.536,A -85,B 0,C 180,E1 -12526.076,E2 -12526.076} C_VEL
LIN {X 0,Y 374.488,Z 436.19,A -85,B 0,C 180,E1 -12526.952,E2 -12526.952} C_VEL
LIN {X 0,Y 371.974,Z 433.546,A -85,B 0,C 180,E1 -12528.368,E2 -12528.368} C_VEL
LIN {X 0,Y 369.528,Z 430.284,A -85,B 0,C 180,E1 -12529.768,E2 -12529.768} C_VEL
LIN {X 0,Y 369.196,Z 427.829,A -85,B 0,C 180,E1 -12530.607,E2 -12530.607} C_VEL
LIN {X 0,Y 370.046,Z 421.609,A -85,B 0,C 180,E1 -12532.324,E2 -12532.324} C_VEL
LIN {X 0,Y 371.1,Z 413.85,A -85,B 0,C 180,E1 -12534.027,E2 -12534.027} C_VEL
LIN {X 0,Y 372.155,Z 405.707,A -85,B 0,C 180,E1 -12535.461,E2 -12535.461} C_VEL
LIN {X 0,Y 373.311,Z 395.902,A -85,B 0,C 180,E1 -12536.86,E2 -12536.86} C_VEL
LIN {X 0,Y 374.486,Z 386.155,A -85,B 0,C 180,E1 -12537.98,E2 -12537.98} C_VEL
LIN {X 0,Y 375.502,Z 375.595,A -85,B 0,C 180,E1 -12538.965,E2 -12538.965} C_VEL
LIN {X 0,Y 376.305,Z 363.977,A -85,B 0,C 180,E1 -12539.818,E2 -12539.818} C_VEL
LIN {X 0,Y 377.197,Z 350.658,A -85,B 0,C 180,E1 -12540.517,E2 -12540.517} C_VEL
LIN {X 0,Y 377.679,Z 338.229,A -85,B 0,C 180,E1 -12540.96,E2 -12540.96} C_VEL
LIN {X 0,Y 379.253,Z 254.59,A -85,B 0,C 180,E1 -12542.598,E2 -12542.598} C_VEL
LIN {X 0,Y 376.895,Z 245.72,A -85,B 0,C 180,E1 -12542.952,E2 -12542.952} C_VEL
LIN {X 0,Y 370.581,Z 230.628,A -85,B 0,C 180,E1 -12543.774,E2 -12543.774} C_VEL
LIN {X 0,Y 368.942,Z 223.529,A -85,B 0,C 180,E1 -12545.812,E2 -12545.812} C_VEL
LIN {X 0,Y 368.903,Z 223.538,A -85,B 0,C 180,E1 -12548.951,E2 -12548.951} C_VEL
LIN {X 0,Y 368.903,Z 223.54,A -85,B 0,C 180,E1 -12552.013,E2 -12552.013} C_VEL
LIN {X 0,Y 368.942,Z 223.527,A -85,B 0,C 180,E1 -12555.185,E2 -12555.185} C_VEL
LIN {X 0,Y 368.931,Z 223.532,A -85,B 0,C 180,E1 -12558.184,E2 -12558.184} C_VEL
LIN {X 0,Y 368.9,Z 223.533,A -85,B 0,C 180,E1 -12561.358,E2 -12561.358} C_VEL
LIN {X 0,Y 368.923,Z 223.528,A -85,B 0,C 180,E1 -12565.145,E2 -12565.145} C_VEL
LIN {X 0,Y 368.915,Z 223.525,A -85,B 0,C 180,E1 -12569.045,E2 -12569.045} C_VEL
LIN {X 0,Y 368.964,Z 223.526,A -85,B 0,C 180,E1 -12571.562,E2 -12571.562} C_VEL
LIN {X 0,Y 368.981,Z 223.524,A -85,B 0,C 180,E1 -12574.018,E2 -12574.018} C_VEL
LIN {X 0,Y 368.901,Z 223.531,A -85,B 0,C 180,E1 -12577.603,E2 -12577.603} C_VEL
LIN {X 0,Y 368.94,Z 223.521,A -85,B 0,C 180,E1 -12581.105,E2 -12581.105} C_VEL
LIN {X 0,Y 368.976,Z 223.514,A -85,B 0,C 180,E1 -12584.534,E2 -12584.534} C_VEL
LIN {X 0,Y 368.979,Z 223.519,A -85,B 0,C 180,E1 -12587.906,E2 -12587.906} C_VEL
LIN {X 0,Y 369.144,Z 223.501,A -85,B 0,C 180,E1 -12591.869,E2 -12591.869} C_VEL
LIN {X 0,Y 369.118,Z 223.5,A -85,B 0,C 180,E1 -12594.537,E2 -12594.537} C_VEL
LIN {X 0,Y 369.288,Z 223.476,A -85,B 0,C 180,E1 -12597.819,E2 -12597.819} C_VEL
LIN {X 0,Y 369.43,Z 223.464,A -85,B 0,C 180,E1 -12600,E2 -12600} C_VEL
LIN {X 0,Y 369.288,Z 223.479,A -85,B 0,C 180,E1 -12602.181,E2 -12602.181} C_VEL
LIN {X 0,Y 369.151,Z 223.5,A -85,B 0,C 180,E1 -12606.559,E2 -12606.559} C_VEL
LIN {X 0,Y 369.04,Z 223.513,A -85,B 0,C 180,E1 -12609.869,E2 -12609.869} C_VEL
LIN {X 0,Y 369.015,Z 223.515,A -85,B 0,C 180,E1 -12613.772,E2 -12613.772} C_VEL
LIN {X 0,Y 368.971,Z 223.518,A -85,B 0,C 180,E1 -12617.744,E2 -12617.744} C_VEL
LIN {X 0,Y 368.889,Z 223.527,A -85,B 0,C 180,E1 -12621.222,E2 -12621.222} C_VEL
LIN {X 0,Y 368.9,Z 223.531,A -85,B 0,C 180,E1 -12623.879,E2 -12623.879} C_VEL
LIN {X 0,Y 368.851,Z 223.539,A -85,B 0,C 180,E1 -12627.212,E2 -12627.212} C_VEL
LIN {X 0,Y 368.877,Z 223.528,A -85,B 0,C 180,E1 -12629.694,E2 -12629.694} C_VEL
LIN {X 0,Y 368.879,Z 223.527,A -85,B 0,C 180,E1 -12633.54,E2 -12633.54} C_VEL
LIN {X 0,Y 368.882,Z 223.526,A -85,B 0,C 180,E1 -12636.856,E2 -12636.856} C_VEL
LIN {X 0,Y 368.897,Z 223.528,A -85,B 0,C 180,E1 -12640.372,E2 -12640.372} C_VEL
LIN {X 0,Y 368.871,Z 223.535,A -85,B 0,C 180,E1 -12643.617,E2 -12643.617} C_VEL
LIN {X 0,Y 368.876,Z 223.535,A -85,B 0,C 180,E1 -12646.697,E2 -12646.697} C_VEL
LIN {X 0,Y 368.877,Z 223.534,A -85,B 0,C 180,E1 -12649.65,E2 -12649.65} C_VEL
LIN {X 0,Y 368.894,Z 223.535,A -85,B 0,C 180,E1 -12653.146,E2 -12653.146} C_VEL
LIN {X 0,Y 368.893,Z 223.533,A -85,B 0,C 180,E1 -12656.463,E2 -12656.463} C_VEL
LIN {X 0,Y 368.936,Z 223.57,A -85,B 0,C 180,E1 -12658.49,E2 -12658.49} C_VEL
LIN {X 0,Y 371.998,Z 236.449,A -85,B 0,C 180,E1 -12661.816,E2 -12661.816} C_VEL
LIN {X 0,Y 373.764,Z 245.721,A -85,B 0,C 180,E1 -12664.077,E2 -12664.077} C_VEL
LIN {X 0,Y 372.438,Z 258.964,A -85,B 0,C 180,E1 -12666.948,E2 -12666.948} C_VEL
LIN {X 0,Y 372.227,Z 261.184,A -85,B 0,C 180,E1 -12667.426,E2 -12667.426} C_VEL
LIN {X 0,Y 376.762,Z 284.893,A -85,B 0,C 180,E1 -12668.264,E2 -12668.264} C_VEL
LIN {X 0,Y 378.575,Z 297.85,A -85,B 0,C 180,E1 -12668.656,E2 -12668.656} C_VEL
LIN {X 0,Y 377.269,Z 370.657,A -85,B 0,C 180,E1 -12670.089,E2 -12670.089} C_VEL
LIN {X 0,Y 376.523,Z 383.677,A -85,B 0,C 180,E1 -12670.545,E2 -12670.545} C_VEL
LIN {X 0,Y 375.392,Z 396.823,A -85,B 0,C 180,E1 -12671.229,E2 -12671.229} C_VEL
LIN {X 0,Y 374.284,Z 408.677,A -85,B 0,C 180,E1 -12672.092,E2 -12672.092} C_VEL
LIN {X 0,Y 373.027,Z 420.076,A -85,B 0,C 180,E1 -12673.161,E2 -12673.161} C_VEL
LIN {X 0,Y 371.818,Z 430.378,A -85,B 0,C 180,E1 -12674.374,E2 -12674.374} C_VEL
LIN {X 0,Y 370.705,Z 439.662,A -85,B 0,C 180,E1 -12675.731,E2 -12675.731} C_VEL
LIN {X 0,Y 369.59,Z 448.684,A -85,B 0,C 180,E1 -12677.368,E2 -12677.368} C_VEL
LIN {X 0,Y 368.646,Z 455.978,A -85,B 0,C 180,E1 -12679.009,E2 -12679.009} C_VEL
LIN {X 0,Y 368.09,Z 461.847,A -85,B 0,C 180,E1 -12680.659,E2 -12680.659} C_VEL
LIN {X 0,Y 367.699,Z 466.491,A -85,B 0,C 180,E1 -12682.31,E2 -12682.31} C_VEL
LIN {X 0,Y 367.511,Z 470.003,A -85,B 0,C 180,E1 -12683.94,E2 -12683.94} C_VEL
LIN {X 0,Y 367.455,Z 472.605,A -85,B 0,C 180,E1 -12685.611,E2 -12685.611} C_VEL
LIN {X 0,Y 367.404,Z 473.81,A -85,B 0,C 180,E1 -12686.708,E2 -12686.708} C_VEL
LIN {X 0,Y 367.538,Z 474.954,A -85,B 0,C 180,E1 -12688.902,E2 -12688.902} C_VEL
LIN {X 0,Y 367.544,Z 474.941,A -85,B 0,C 180,E1 -12689.998,E2 -12689.998} C_VEL
LIN {X 0,Y 367.56,Z 474.538,A -85,B 0,C 180,E1 -12691.093,E2 -12691.093} C_VEL
LIN {X 0,Y 367.493,Z 473.691,A -85,B 0,C 180,E1 -12692.19,E2 -12692.19} C_VEL
LIN {X 0,Y 367.506,Z 470.773,A -85,B 0,C 180,E1 -12694.385,E2 -12694.385} C_VEL
LIN {X 0,Y 367.521,Z 467.317,A -85,B 0,C 180,E1 -12696.075,E2 -12696.075} C_VEL
LIN {X 0,Y 367.688,Z 462.959,A -85,B 0,C 180,E1 -12697.686,E2 -12697.686} C_VEL
LIN {X 0,Y 367.967,Z 457.287,A -85,B 0,C 180,E1 -12699.34,E2 -12699.34} C_VEL
LIN {X 0,Y 368.438,Z 450.182,A -85,B 0,C 180,E1 -12700.993,E2 -12700.993} C_VEL
LIN {X 0,Y 369.264,Z 441.294,A -85,B 0,C 180,E1 -12702.64,E2 -12702.64} C_VEL
LIN {X 0,Y 370.074,Z 431.169,A -85,B 0,C 180,E1 -12704.149,E2 -12704.149} C_VEL
LIN {X 0,Y 370.936,Z 420.8,A -85,B 0,C 180,E1 -12705.378,E2 -12705.378} C_VEL
LIN {X 0,Y 371.857,Z 409.293,A -85,B 0,C 180,E1 -12706.465,E2 -12706.465} C_VEL
LIN {X 0,Y 372.747,Z 397.301,A -85,B 0,C 180,E1 -12707.342,E2 -12707.342} C_VEL
LIN {X 0,Y 373.483,Z 384.735,A -85,B 0,C 180,E1 -12708.014,E2 -12708.014} C_VEL
LIN {X 0,Y 374.122,Z 371.846,A -85,B 0,C 180,E1 -12708.478,E2 -12708.478} C_VEL
LIN {X 0,Y 374.802,Z 328.88,A -85,B 0,C 180,E1 -12709.33,E2 -12709.33} C_VEL
LIN {X 0,Y 375.077,Z 294.889,A -85,B 0,C 180,E1 -12709.986,E2 -12709.986} C_VEL
LIN {X 0,Y 370.626,Z 261.83,A -85,B 0,C 180,E1 -12710.86,E2 -12710.86} C_VEL
LIN {X 0,Y 371.953,Z 244.22,A -85,B 0,C 180,E1 -12714.558,E2 -12714.558} C_VEL
LIN {X 0,Y 372.147,Z 239.765,A -85,B 0,C 180,E1 -12715.508,E2 -12715.508} C_VEL
LIN {X 0,Y 369.786,Z 227.331,A -85,B 0,C 180,E1 -12718.363,E2 -12718.363} C_VEL
LIN {X 0,Y 368.947,Z 223.528,A -85,B 0,C 180,E1 -12719.278,E2 -12719.278} C_VEL
LIN {X 0,Y 368.88,Z 223.532,A -85,B 0,C 180,E1 -12723.039,E2 -12723.039} C_VEL
LIN {X 0,Y 368.897,Z 223.534,A -85,B 0,C 180,E1 -12726.192,E2 -12726.192} C_VEL
LIN {X 0,Y 368.879,Z 223.532,A -85,B 0,C 180,E1 -12728.949,E2 -12728.949} C_VEL
LIN {X 0,Y 368.856,Z 223.54,A -85,B 0,C 180,E1 -12732.005,E2 -12732.005} C_VEL
LIN {X 0,Y 368.923,Z 223.528,A -85,B 0,C 180,E1 -12735.182,E2 -12735.182} C_VEL
LIN {X 0,Y 368.915,Z 223.53,A -85,B 0,C 180,E1 -12738.182,E2 -12738.182} C_VEL
LIN {X 0,Y 368.879,Z 223.535,A -85,B 0,C 180,E1 -12741.355,E2 -12741.355} C_VEL
LIN {X 0,Y 368.9,Z 223.531,A -85,B 0,C 180,E1 -12745.142,E2 -12745.142} C_VEL
LIN {X 0,Y 368.892,Z 223.532,A -85,B 0,C 180,E1 -12749.043,E2 -12749.043} C_VEL
LIN {X 0,Y 368.94,Z 223.531,A -85,B 0,C 180,E1 -12751.561,E2 -12751.561} C_VEL
LIN {X 0,Y 368.919,Z 223.531,A -85,B 0,C 180,E1 -12755.222,E2 -12755.222} C_VEL
LIN {X 0,Y 368.947,Z 223.526,A -85,B 0,C 180,E1 -12758.949,E2 -12758.949} C_VEL
LIN {X 0,Y 368.946,Z 223.524,A -85,B 0,C 180,E1 -12762.255,E2 -12762.255} C_VEL
LIN {X 0,Y 368.99,Z 223.518,A -85,B 0,C 180,E1 -12766.226,E2 -12766.226} C_VEL
LIN {X 0,Y 369.025,Z 223.514,A -85,B 0,C 180,E1 -12770.131,E2 -12770.131} C_VEL
LIN {X 0,Y 369.144,Z 223.499,A -85,B 0,C 180,E1 -12772.341,E2 -12772.341} C_VEL
LIN {X 0,Y 369.101,Z 223.506,A -85,B 0,C 180,E1 -12774.537,E2 -12774.537} C_VEL
LIN {X 0,Y 369.267,Z 223.484,A -85,B 0,C 180,E1 -12777.819,E2 -12777.819} C_VEL
LIN {X 0,Y 369.406,Z 223.467,A -85,B 0,C 180,E1 -12780,E2 -12780} C_VEL
LIN {X 0,Y 369.263,Z 223.485,A -85,B 0,C 180,E1 -12782.182,E2 -12782.182} C_VEL
LIN {X 0,Y 369.14,Z 223.502,A -85,B 0,C 180,E1 -12786.654,E2 -12786.654} C_VEL
LIN {X 0,Y 369.02,Z 223.515,A -85,B 0,C 180,E1 -12789.87,E2 -12789.87} C_VEL
LIN {X 0,Y 368.99,Z 223.518,A -85,B 0,C 180,E1 -12793.774,E2 -12793.774} C_VEL
LIN {X 0,Y 368.957,Z 223.523,A -85,B 0,C 180,E1 -12797.771,E2 -12797.771} C_VEL
LIN {X 0,Y 368.865,Z 223.535,A -85,B 0,C 180,E1 -12801.224,E2 -12801.224} C_VEL
LIN {X 0,Y 368.912,Z 223.533,A -85,B 0,C 180,E1 -12804.779,E2 -12804.779} C_VEL
LIN {X 0,Y 368.928,Z 223.527,A -85,B 0,C 180,E1 -12807.207,E2 -12807.207} C_VEL
LIN {X 0,Y 368.882,Z 223.532,A -85,B 0,C 180,E1 -12809.694,E2 -12809.694} C_VEL
LIN {X 0,Y 368.86,Z 223.536,A -85,B 0,C 180,E1 -12813.047,E2 -12813.047} C_VEL
LIN {X 0,Y 368.882,Z 223.536,A -85,B 0,C 180,E1 -12816.201,E2 -12816.201} C_VEL
LIN {X 0,Y 368.874,Z 223.534,A -85,B 0,C 180,E1 -12818.957,E2 -12818.957} C_VEL
LIN {X 0,Y 368.922,Z 223.53,A -85,B 0,C 180,E1 -12822.026,E2 -12822.026} C_VEL
LIN {X 0,Y 368.893,Z 223.53,A -85,B 0,C 180,E1 -12825.186,E2 -12825.186} C_VEL
LIN {X 0,Y 368.858,Z 223.541,A -85,B 0,C 180,E1 -12828.182,E2 -12828.182} C_VEL
LIN {X 0,Y 368.887,Z 223.532,A -85,B 0,C 180,E1 -12831.365,E2 -12831.365} C_VEL
LIN {X 0,Y 368.918,Z 223.527,A -85,B 0,C 180,E1 -12835.151,E2 -12835.151} C_VEL
LIN {X 0,Y 368.915,Z 223.528,A -85,B 0,C 180,E1 -12839.051,E2 -12839.051} C_VEL
LIN {X 0,Y 368.952,Z 223.523,A -85,B 0,C 180,E1 -12842.801,E2 -12842.801} C_VEL
LIN {X 0,Y 368.925,Z 223.53,A -85,B 0,C 180,E1 -12846.121,E2 -12846.121} C_VEL
LIN {X 0,Y 368.93,Z 223.531,A -85,B 0,C 180,E1 -12849.951,E2 -12849.951} C_VEL
LIN {X 0,Y 368.964,Z 223.524,A -85,B 0,C 180,E1 -12853.402,E2 -12853.402} C_VEL
LIN {X 0,Y 369.056,Z 223.51,A -85,B 0,C 180,E1 -12856.794,E2 -12856.794} C_VEL
LIN {X 0,Y 369.051,Z 223.636,A -85,B 0,C 180,E1 -12858.538,E2 -12858.538} C_VEL
LIN {X 0,Y 370.319,Z 230.168,A -85,B 0,C 180,E1 -12860.213,E2 -12860.213} C_VEL
LIN {X 0,Y 373.06,Z 239.459,A -85,B 0,C 180,E1 -12860.54,E2 -12860.54} C_VEL
LIN {X 0,Y 375.75,Z 254.022,A -85,B 0,C 180,E1 -12860.957,E2 -12860.957} C_VEL
LIN {X 0,Y 374.319,Z 337.208,A -85,B 0,C 180,E1 -12862.552,E2 -12862.552} C_VEL
LIN {X 0,Y 373.864,Z 350.467,A -85,B 0,C 180,E1 -12863.018,E2 -12863.018} C_VEL
LIN {X 0,Y 373.356,Z 362.564,A -85,B 0,C 180,E1 -12863.653,E2 -12863.653} C_VEL
LIN {X 0,Y 372.844,Z 373.944,A -85,B 0,C 180,E1 -12864.459,E2 -12864.459} C_VEL
LIN {X 0,Y 371.825,Z 385.723,A -85,B 0,C 180,E1 -12865.531,E2 -12865.531} C_VEL
LIN {X 0,Y 370.96,Z 396.222,A -85,B 0,C 180,E1 -12866.744,E2 -12866.744} C_VEL
LIN {X 0,Y 370.123,Z 405.697,A -85,B 0,C 180,E1 -12868.098,E2 -12868.098} C_VEL
